// ---- analog_input/voltage/EL3164.TcPOU
(**
This function block abstracts the Beckhoff EtherCAT terminal EL3164 (0…10 V, 16 Bit)
*)
FUNCTION_BLOCK EL3164 IMPLEMENTS I_terminal_execution
VAR_INPUT
END_VAR
VAR_OUTPUT
	AI_Voltage_channel_1 		: I_AI_Voltage := _ar_channels[1];
	AI_Voltage_channel_2 		: I_AI_Voltage := _ar_channels[2];
	AI_Voltage_channel_3 		: I_AI_Voltage := _ar_channels[3];
	AI_Voltage_channel_4 		: I_AI_Voltage := _ar_channels[4];
	AI_percent_channe_1			: I_AI_percentage := _ar_channels[1];
	AI_percent_channe_2			: I_AI_percentage := _ar_channels[2];
	AI_percent_channe_3			: I_AI_percentage := _ar_channels[3];
	AI_percent_channe_4			: I_AI_percentage := _ar_channels[4];
END_VAR
VAR
// == IO Mapping ==============================================================
// The channel status Limits 1 and 2 have to be defined as BYTE since they are 
// of BIT2 in the terminal, but there is no such datatype in the PLC.

	WcState_WcState			AT%I*: BOOL;
	InfoData_State			AT%I*: UINT;
	InfoData_AdsAddr_netId  AT%I*: AMSNETID;
	InfoData_AdsAddr_port 	AT%I*: WORD;
	
	// Channel 1
	AI_Standard_Channel_1_Value        			AT%I*: INT;	
	AI_Standard_Channel_1_Status_Underrange   	AT%I*: BOOL;
	AI_Standard_Channel_1_Status_Overrange   	AT%I*: BOOL;
	AI_Standard_Channel_1_Status_Limit_1   		AT%I*: BYTE;
	AI_Standard_Channel_1_Status_Limit_2   		AT%I*: BYTE;
	AI_Standard_Channel_1_Status_Error   		AT%I*: BOOL;
	AI_Standard_Channel_1_Status_Sync_error   	AT%I*: BOOL;
	AI_Standard_Channel_1_Status_TxPDO_State   	AT%I*: BOOL;
	AI_Standard_Channel_1_Status_TxPDO_Toggle   AT%I*: BOOL;

	// Channel 2
	AI_Standard_Channel_2_Value        			AT%I*: INT;	
	AI_Standard_Channel_2_Status_Underrange   	AT%I*: BOOL;
	AI_Standard_Channel_2_Status_Overrange   	AT%I*: BOOL;
	AI_Standard_Channel_2_Status_Limit_1   		AT%I*: BYTE;
	AI_Standard_Channel_2_Status_Limit_2   		AT%I*: BYTE;
	AI_Standard_Channel_2_Status_Error   		AT%I*: BOOL;
	AI_Standard_Channel_2_Status_Sync_error   	AT%I*: BOOL;
	AI_Standard_Channel_2_Status_TxPDO_State   	AT%I*: BOOL;
	AI_Standard_Channel_2_Status_TxPDO_Toggle   AT%I*: BOOL;
	
	// Channel 3
	AI_Standard_Channel_3_Value        			AT%I*: INT;	
	AI_Standard_Channel_3_Status_Underrange   	AT%I*: BOOL;
	AI_Standard_Channel_3_Status_Overrange   	AT%I*: BOOL;
	AI_Standard_Channel_3_Status_Limit_1   		AT%I*: BYTE;
	AI_Standard_Channel_3_Status_Limit_2   		AT%I*: BYTE;
	AI_Standard_Channel_3_Status_Error   		AT%I*: BOOL;
	AI_Standard_Channel_3_Status_Sync_error   	AT%I*: BOOL;
	AI_Standard_Channel_3_Status_TxPDO_State   	AT%I*: BOOL;
	AI_Standard_Channel_3_Status_TxPDO_Toggle   AT%I*: BOOL;
	
	// Channel 4
	AI_Standard_Channel_4_Value        			AT%I*: INT;	
	AI_Standard_Channel_4_Status_Underrange   	AT%I*: BOOL;
	AI_Standard_Channel_4_Status_Overrange   	AT%I*: BOOL;
	AI_Standard_Channel_4_Status_Limit_1   		AT%I*: BYTE;  
	AI_Standard_Channel_4_Status_Limit_2   		AT%I*: BYTE;
	AI_Standard_Channel_4_Status_Error   		AT%I*: BOOL;
	AI_Standard_Channel_4_Status_Sync_error   	AT%I*: BOOL;
	AI_Standard_Channel_4_Status_TxPDO_State   	AT%I*: BOOL;
	AI_Standard_Channel_4_Status_TxPDO_Toggle   AT%I*: BOOL;
// ============================================================================

    _ar_channels : ARRAY[1..NUMBER_OF_CHANNELS] OF AI_Voltage_Channel[
		(adc_min:=ADC_MIN, adc_max:=ADC_MAX, physical_min:=PHYSICAL_MIN, physical_max:=PHYSICAL_MAX,channel_number:=1),
		(adc_min:=ADC_MIN, adc_max:=ADC_MAX, physical_min:=PHYSICAL_MIN, physical_max:=PHYSICAL_MAX,channel_number:=2),
		(adc_min:=ADC_MIN, adc_max:=ADC_MAX, physical_min:=PHYSICAL_MIN, physical_max:=PHYSICAL_MAX,channel_number:=3),
		(adc_min:=ADC_MIN, adc_max:=ADC_MAX, physical_min:=PHYSICAL_MIN, physical_max:=PHYSICAL_MAX,channel_number:=4)
    ];
    
	// ===============================================================================
	// CoE handling  
	// ==============
    _I_CoE_com_handler      : I_CoE_communication_handler;
    _CoE_prop_handler       : CoE_property_handler;
    // ====  CoE properties  ===========
	_p_DeviceName 			: CoE_property_string(Index:=16#1008 , SubIndex:=0, writable:=FALSE, propertyType:=0, pollingInterval:=T#5S);
	_p_DeviceType 			: CoE_property_udint(Index:=16#1000 , SubIndex:=0, writable:=FALSE, propertyType:=0, pollingInterval:=T#5S);
	_p_ProductCode 			: CoE_property_udint(Index:=16#1018 , SubIndex:=2, writable:=FALSE, propertyType:=0, pollingInterval:=T#5S);
	_p_Revision 			: CoE_property_udint(Index:=16#1018 , SubIndex:=3, writable:=FALSE, propertyType:=0, pollingInterval:=T#5S);
	_p_SerialNumber 		: CoE_property_udint(Index:=16#1018 , SubIndex:=4, writable:=FALSE, propertyType:=0, pollingInterval:=T#5S);
	_p_SoftwareVersion		: CoE_property_string(Index:=16#100A , SubIndex:=0, writable:=FALSE, propertyType:=0, pollingInterval:=T#5S);
	_p_VendorId 			: CoE_property_udint(Index:=16#1018 , SubIndex:=1, writable:=FALSE, propertyType:=0, pollingInterval:=T#5S);
	_p_HardwareVersion		: CoE_property_string(Index:=16#1009 , SubIndex:=0, writable:=FALSE, propertyType:=0, pollingInterval:=T#5S);
	// ==============
	_properties  : ARRAY[1..8]OF I_CoE_property:=[
		_p_DeviceName, _p_DeviceType, _p_ProductCode, _p_Revision, _p_SerialNumber, 
		_p_SoftwareVersion, _p_VendorId, _p_HardwareVersion
	];
	// ===============================================================================
    
    
	_I_InterfaceManager : I_InterfaceManager;
	_terminal_name      : STRING;
    errId               : HAL_ErrorEnum;
	_InitState          : INT;
    neg_wcState: f_trig;
    _j:INT;
	_terminal_id: UINT;

END_VAR
VAR CONSTANT
	ADC_MIN        	: INT:=0;
	ADC_MAX        	: INT:=32767;
	PHYSICAL_MIN 	: INT:=0;
	PHYSICAL_MAX 	: INT:=10;
	
    HARDWARE_REVSION : UINT:=19;
    NUMBER_OF_CHANNELS : INT:=4;
END_VAR


// Channel 1
_ar_channels[1].wcState							:= WcState_WcState;
_ar_channels[1].terminal_value                  := AI_Standard_Channel_1_Value;
_ar_channels[1].io_status_Underrange            := AI_Standard_Channel_1_Status_Underrange;
_ar_channels[1].io_status_Overrange             := AI_Standard_Channel_1_Status_Overrange;
_ar_channels[1].io_status_Limit_1_greater_value := AI_Standard_Channel_1_Status_Limit_1.0;
_ar_channels[1].io_status_Limit_1_smaller_value := AI_Standard_Channel_1_Status_Limit_1.1;
_ar_channels[1].io_status_Limit_2_greater_value := AI_Standard_Channel_1_Status_Limit_2.0;
_ar_channels[1].io_status_Limit_2_smaller_value := AI_Standard_Channel_1_Status_Limit_2.1;
_ar_channels[1].io_status_Error                 := AI_Standard_Channel_1_Status_Error;
_ar_channels[1].io_status_Sync_error            := AI_Standard_Channel_1_Status_Sync_error;
_ar_channels[1].io_status_TxPDO_State           := AI_Standard_Channel_1_Status_TxPDO_State;
_ar_channels[1].io_status_TxPDO_Toggle          := AI_Standard_Channel_1_Status_TxPDO_Toggle;

// Channel 2
_ar_channels[2].wcState                         := WcState_WcState;
_ar_channels[2].terminal_value                  := AI_Standard_Channel_2_Value;
_ar_channels[2].io_status_Underrange            := AI_Standard_Channel_2_Status_Underrange;
_ar_channels[2].io_status_Overrange             := AI_Standard_Channel_2_Status_Overrange;
_ar_channels[2].io_status_Limit_1_greater_value := AI_Standard_Channel_2_Status_Limit_1.0;
_ar_channels[2].io_status_Limit_1_smaller_value := AI_Standard_Channel_2_Status_Limit_1.1;
_ar_channels[2].io_status_Limit_2_greater_value := AI_Standard_Channel_2_Status_Limit_2.0;
_ar_channels[2].io_status_Limit_2_smaller_value := AI_Standard_Channel_2_Status_Limit_2.1;
_ar_channels[2].io_status_Error                 := AI_Standard_Channel_2_Status_Error;
_ar_channels[2].io_status_Sync_error            := AI_Standard_Channel_2_Status_Sync_error;
_ar_channels[2].io_status_TxPDO_State           := AI_Standard_Channel_2_Status_TxPDO_State;
_ar_channels[2].io_status_TxPDO_Toggle          := AI_Standard_Channel_2_Status_TxPDO_Toggle;

// Channel 3
_ar_channels[3].wcState                         := WcState_WcState;
_ar_channels[3].terminal_value                  := AI_Standard_Channel_3_Value;
_ar_channels[3].io_status_Underrange            := AI_Standard_Channel_3_Status_Underrange;
_ar_channels[3].io_status_Overrange             := AI_Standard_Channel_3_Status_Overrange;
_ar_channels[3].io_status_Limit_1_greater_value := AI_Standard_Channel_3_Status_Limit_1.0;
_ar_channels[3].io_status_Limit_1_smaller_value := AI_Standard_Channel_3_Status_Limit_1.1;
_ar_channels[3].io_status_Limit_2_greater_value := AI_Standard_Channel_3_Status_Limit_2.0;
_ar_channels[3].io_status_Limit_2_smaller_value := AI_Standard_Channel_3_Status_Limit_2.1;
_ar_channels[3].io_status_Error                 := AI_Standard_Channel_3_Status_Error;
_ar_channels[3].io_status_Sync_error            := AI_Standard_Channel_3_Status_Sync_error;
_ar_channels[3].io_status_TxPDO_State           := AI_Standard_Channel_3_Status_TxPDO_State;
_ar_channels[3].io_status_TxPDO_Toggle          := AI_Standard_Channel_3_Status_TxPDO_Toggle;

// Channel 4
_ar_channels[4].wcState                         := WcState_WcState;
_ar_channels[4].terminal_value                  := AI_Standard_Channel_4_Value;
_ar_channels[4].io_status_Underrange            := AI_Standard_Channel_4_Status_Underrange;
_ar_channels[4].io_status_Overrange             := AI_Standard_Channel_4_Status_Overrange;
_ar_channels[4].io_status_Limit_1_greater_value := AI_Standard_Channel_4_Status_Limit_1.0;
_ar_channels[4].io_status_Limit_1_smaller_value := AI_Standard_Channel_4_Status_Limit_1.1;
_ar_channels[4].io_status_Limit_2_greater_value := AI_Standard_Channel_4_Status_Limit_2.0;
_ar_channels[4].io_status_Limit_2_smaller_value := AI_Standard_Channel_4_Status_Limit_2.1;
_ar_channels[4].io_status_Error                 := AI_Standard_Channel_4_Status_Error;
_ar_channels[4].io_status_Sync_error            := AI_Standard_Channel_4_Status_Sync_error;
_ar_channels[4].io_status_TxPDO_State           := AI_Standard_Channel_4_Status_TxPDO_State;
_ar_channels[4].io_status_TxPDO_Toggle          := AI_Standard_Channel_4_Status_TxPDO_Toggle;


IF  _I_InterfaceManager <> 0 AND 
    _I_CoE_com_handler <> 0
THEN
    FOR _j:=1 TO NUMBER_OF_CHANNELS DO
        // should be possible to get rid of the address input 
        _ar_channels[_j](terminal_address:=InfoData_AdsAddr_port, CoE_communication_handler:=_I_CoE_com_handler);
    END_FOR
    
    _CoE_prop_handler(terminal_address:=InfoData_AdsAddr_port, CoE_communication_handler:=_I_CoE_com_handler, CoE_properties:=_properties);

    neg_wcState(CLK:=WcState_WcState);
    IF neg_wcState.Q THEN
        ;
    END_IF
END_IF

METHOD FB_init : BOOL
VAR_INPUT
	bInitRetains : BOOL; // if TRUE, the retain variables are initialized (warm start / cold start)
	bInCopyCode : BOOL;  // if TRUE, the instance afterwards gets moved into the copy code (online change)
	CoE_communication_handler   : I_CoE_communication_handler;
	InterfaceManager            : I_InterfaceManager;
	name                        : STRING;
END_VAR

_I_CoE_com_handler := CoE_communication_handler;

FOR _j:=1 TO NUMBER_OF_CHANNELS DO
    _ar_channels[_j].CoE_communication_handler := CoE_communication_handler;
END_FOR

_terminal_name := name;
_I_InterfaceManager := InterfaceManager;

// register  terminal and all channel interfaces
IF InterfaceManager <> 0 THEN
    _I_InterfaceManager.register_terminal(terminal_name:=_terminal_name , errId=>errId , terminalId=>_terminal_id);
    
    FOR _j:=1 TO NUMBER_OF_CHANNELS DO
        _ar_channels[_j].register_channel(terminalId:=_terminal_id , I_interface_manager:=_I_InterfaceManager , errId=>errId );
        IF errId <> HAL_ErrorEnum.no_error THEN
            ;  // ToDo: add logging or Error handling 
        END_IF 
    END_FOR
END_IF
END_METHOD

METHOD run : BOOL
THIS^();
END_METHOD

END_FUNCTION_BLOCK

// ---- analog_input/_internal/AI_Voltage_Channel.TcPOU
FUNCTION_BLOCK AI_Voltage_Channel IMPLEMENTS I_AI_Voltage, I_AI_percentage
VAR_INPUT
	terminal_address		    : WORD;
	CoE_communication_handler	: I_CoE_communication_handler;
END_VAR
VAR_OUTPUT
END_VAR
VAR
	_adc_min        : INT;
    _adc_max        : INT;
	_physical_min 	: INT;
	_physical_max 	: INT;
	_channel_number : UsINT;
	_rValue			: REAL;
	_wcState		: BOOL;
	
	// ===============================================================================
	// CoE handling  
    // ==============
    _CoE_prop_handler      : CoE_property_handler;
    _CoE_channel_offset     : INT;
    index_1 				: WORD:= 16#8000 + INT_TO_WORD(_CoE_channel_offset);	
    // ====  CoE properties  ===========
	_p_Enable_user_scale    		: CoE_property_bool(Index:=index_1 , SubIndex:=1, writable:=TRUE, propertyType:=0, pollingInterval:=T#5S);
	_p_Presentation 				: CoE_property_usint(Index:=index_1 , SubIndex:=2, writable:=TRUE, propertyType:=0, pollingInterval:=T#5S);			// DT0800EN03
	_p_Watchdog 					: CoE_property_usint(Index:=index_1 , SubIndex:=5, writable:=TRUE, propertyType:=0, pollingInterval:=T#5S);			// DT0801EN02
	_p_Enable_user_calibration  	: CoE_property_bool(Index:=index_1 , SubIndex:=7, writable:=TRUE, propertyType:=0, pollingInterval:=T#5S);
	_p_Enable_vendor_calibration    : CoE_property_bool(Index:=index_1 , SubIndex:=8, writable:=TRUE, propertyType:=0, pollingInterval:=T#5S);
	_p_Offset   					: CoE_property_int(Index:=index_1 , SubIndex:=17, writable:=TRUE, propertyType:=0, pollingInterval:=T#5S);
	_p_Gain 						: CoE_property_dint(Index:=index_1 , SubIndex:=18, writable:=TRUE, propertyType:=0, pollingInterval:=T#5S);
	_p_Default_output   			: CoE_property_int(Index:=index_1 , SubIndex:=19, writable:=TRUE, propertyType:=0, pollingInterval:=T#5S);
	_p_Default_output_ramp  		: CoE_property_uint(Index:=index_1 , SubIndex:=20, writable:=TRUE, propertyType:=0, pollingInterval:=T#5S);
	_p_User_calibration_offset  	: CoE_property_int(Index:=index_1 , SubIndex:=21, writable:=TRUE, propertyType:=0, pollingInterval:=T#5S);
	_p_User_calibration_gain    	: CoE_property_uint(Index:=index_1 , SubIndex:=22, writable:=TRUE, propertyType:=0, pollingInterval:=T#5S);
	// ==============
	_properties  : ARRAY[1..11]OF I_CoE_property:=[
		_p_Enable_user_scale, _p_Presentation, _p_Watchdog, _p_Enable_user_calibration, _p_Enable_vendor_calibration, _p_Offset,
		_p_Gain, _p_Default_output, _p_Default_output_ramp, _p_User_calibration_offset, _p_User_calibration_gain];
	// ===============================================================================


	//  ====  I_AI_percentage  ====
	_max_value 	: REAL:=10.0;
	_min_value 	: REAL:=0.0;
	_value: REAL;
	
	_errId: HAL_ErrorEnum;
	neg_wcState: f_trig;
END_VAR

// CoE Property handling 
_CoE_prop_handler(terminal_address:=terminal_address, CoE_communication_handler:=CoE_communication_handler, CoE_properties:=_properties);

neg_wcState(CLK:=_wcState);
IF neg_wcState.Q THEN
    ;
END_IF

PROPERTY errId : HAL_ErrorEnum
GET
errId := _errId;
END_GET
END_PROPERTY

METHOD FB_init : BOOL
VAR_INPUT
	bInitRetains 	: BOOL; // if TRUE, the retain variables are initialized (warm start / cold start)
	bInCopyCode 	: BOOL;  // if TRUE, the instance afterwards gets moved into the copy code (online change)
    adc_min         : INT;
    adc_max         : INT;
	physical_min 	: INT;
	physical_max 	: INT;
	channel_number  : UsINT;
END_VAR

VAR
	i: UINT;
END_VAR

_adc_min        := adc_min;
_adc_max        := adc_max;
_physical_min 	:= physical_min;
_physical_max 	:= physical_max;
_channel_number :=channel_number;

CASE channel_number OF
	1:
		_CoE_channel_offset:=16#0;
	2:
		_CoE_channel_offset:=16#10;
	3:
		_CoE_channel_offset:=16#20;
	4:
		_CoE_channel_offset:=16#30;
END_CASE
END_METHOD

METHOD get_Default_output : BOOL
VAR_OUTPUT
	value	: INT;
END_VAR
get_Default_output:=_p_Default_output.get_value(value=>value, errId => );
END_METHOD

METHOD get_Default_output_ramp : BOOL
VAR_OUTPUT
	value	: UINT;
END_VAR
get_Default_output_ramp:=_p_Default_output_ramp.get_value(value=>value, errId => );
END_METHOD

METHOD get_Enable_user_calibration : BOOL
VAR_OUTPUT
	value	: BOOL;
END_VAR
get_Enable_user_calibration:=_p_Enable_user_calibration.get_value(value=>value, errId => );
END_METHOD

METHOD get_Enable_user_scale : BOOL
VAR_OUTPUT
	value	: BOOL;
END_VAR
get_Enable_user_scale:=_p_Enable_user_scale.get_value(value=>value, errId => );
END_METHOD

METHOD get_Enable_vendor_calibration : BOOL
VAR_OUTPUT
	value	: BOOL;
END_VAR
get_Enable_vendor_calibration:=_p_Enable_vendor_calibration.get_value(value=>value, errId => );
END_METHOD

METHOD get_Gain : BOOL
VAR_OUTPUT
	value	: DINT;
END_VAR
get_Gain:=_p_Gain.get_value(value=>value, errId => );
END_METHOD

METHOD get_Offset : BOOL
VAR_OUTPUT
	value	: INT;
END_VAR
get_Offset:=_p_Offset.get_value(value=>value, errId => );
END_METHOD

METHOD get_Presentation : BOOL
VAR_OUTPUT
	value	: ENU_DT0801EN03;
END_VAR

VAR
	tmp: USINT;
END_VAR
get_Presentation:=_p_Presentation.get_value(value=>tmp, errId => );
value:=USINT_TO_INT(tmp);
END_METHOD

METHOD get_User_calibration_gain : BOOL
VAR_OUTPUT
	value	: UINT;
END_VAR
get_User_calibration_gain:=_p_User_calibration_gain.get_value(value=>value, errId => );
END_METHOD

METHOD get_User_calibration_offset : BOOL
VAR_OUTPUT
	value	: INT;
END_VAR
get_User_calibration_offset:=_p_User_calibration_offset.get_value(value=>value, errId => );
END_METHOD

METHOD get_Watchdog : BOOL
VAR_OUTPUT
	value	: ENU_DT0800EN02;
END_VAR

VAR
	tmp: USINT;
END_VAR
get_Watchdog:=_p_Watchdog.get_value(value=>tmp, errId => );
value := USINT_TO_INT(tmp);
END_METHOD

PROPERTY io_status_Error : bool
GET
END_GET
SET
END_SET
END_PROPERTY

PROPERTY io_status_Limit_1_greater_value : bool
GET
END_GET
SET
END_SET
END_PROPERTY

PROPERTY io_status_Limit_1_smaller_value : bool
GET
END_GET
SET
END_SET
END_PROPERTY

PROPERTY io_status_Limit_2_greater_value : bool
GET
END_GET
SET
END_SET
END_PROPERTY

PROPERTY io_status_Limit_2_smaller_value : bool
GET
END_GET
SET
END_SET
END_PROPERTY

PROPERTY io_status_Overrange : bool
GET
END_GET
SET
END_SET
END_PROPERTY

PROPERTY io_status_Sync_error : bool
GET
END_GET
SET
END_SET
END_PROPERTY

PROPERTY io_status_TxPDO_State : bool
GET
END_GET
SET
END_SET
END_PROPERTY

PROPERTY io_status_TxPDO_Toggle : bool
GET
END_GET
SET
END_SET
END_PROPERTY

PROPERTY io_status_Underrange : bool
GET
END_GET
SET
END_SET
END_PROPERTY

PROPERTY max_value : REAL
GET
max_value := _max_value;
END_GET
SET
IF max_value <= 0 THEN
	_max_value := 0.0001;
ELSE
	_max_value := max_value;
END_IF
END_SET
END_PROPERTY

PROPERTY min_value : REAL
GET
min_value := _min_value;
END_GET
SET
_min_value := min_value;
END_SET
END_PROPERTY

METHOD register_channel : BOOL
VAR_INPUT
    terminalId : UINT;
    I_interface_manager : I_interfaceManager;
END_VAR
VAR_OUTPUT
	errId		: HAL_ErrorEnum;
END_VAR
THIS^.register_I_AI_percentage(terminalId:=terminalId , I_interface_manager:=I_interface_manager , errId=>errId );
IF errId = HAL_ErrorEnum.no_error THEN
	THIS^.register_I_AI_Voltage(terminalId:=terminalId , I_interface_manager:=I_interface_manager , errId=>errId );
END_IF
END_METHOD

METHOD register_I_AI_percentage : BOOL
VAR_INPUT
    terminalId : UINT;
    I_interface_manager : I_interfaceManager;
END_VAR
VAR_OUTPUT
	errId		: HAL_ErrorEnum;
END_VAR
register_I_AI_percentage:= I_interface_manager.register_I_AI_Percentage(THIS^, terminalId, channel_number := THIS^._channel_number, errId=>errId);
END_METHOD

METHOD register_I_AI_Voltage : BOOL
VAR_INPUT
    terminalId : UINT;
    I_interface_manager : I_interfaceManager;
END_VAR
VAR_OUTPUT
	errId		: HAL_ErrorEnum;
END_VAR
register_I_AI_Voltage:= I_interface_manager.register_I_AI_Voltage(THIS^, terminalId, channel_number := THIS^._channel_number, errId=>errId);
END_METHOD

PROPERTY rValue : REAL
GET
rValue:=_rValue;
END_GET
SET
IF rValue < DINT_TO_REAL(_physical_min) THEN
	_errId := 6;
ELSIF rValue > DINT_TO_REAL(_physical_max) THEN
	_errId := 7;
ELSE
	_rValue := rValue;
END_IF
END_SET
END_PROPERTY

METHOD set_Default_output : BOOL
VAR_INPUT
	value	: INT;
END_VAR
set_Default_output:=_p_Default_output.set_value(value:=value);
END_METHOD

METHOD set_Default_output_ramp : BOOL
VAR_INPUT
	value	: UINT;
END_VAR
set_Default_output_ramp:=_p_Default_output_ramp.set_value(value:=value);
END_METHOD

METHOD set_Enable_user_calibration : BOOL
VAR_INPUT
	value	: BOOL;
END_VAR
set_Enable_user_calibration:=_p_Enable_user_calibration.set_value(value:=value);
END_METHOD

METHOD set_Enable_user_scale : BOOL
VAR_INPUT
	value	: BOOL;
END_VAR
set_Enable_user_scale:=_p_Enable_user_scale.set_value(value:=value);
END_METHOD

METHOD set_Enable_vendor_calibration : BOOL
VAR_INPUT
	value	: BOOL;
END_VAR
set_Enable_vendor_calibration:=_p_Enable_vendor_calibration.set_value(value:=value);
END_METHOD

METHOD set_Gain : BOOL
VAR_INPUT
	value	: DINT;
END_VAR
set_Gain:=_p_Gain.set_value(value:=value);
END_METHOD

METHOD set_Offset : BOOL
VAR_INPUT
	value	: INT;
END_VAR
set_Offset:=_p_Offset.set_value(value:=value);
END_METHOD

METHOD set_Presentation : BOOL
VAR_INPUT
	value	: ENU_DT0801EN03;
END_VAR
set_Presentation:=_p_Presentation.set_value(value:=INT_TO_USINT(value));
END_METHOD

METHOD set_User_calibration_gain : BOOL
VAR_INPUT
	value	: UINT;
END_VAR
set_User_calibration_gain:=_p_User_calibration_gain.set_value(value:=value);
END_METHOD

METHOD set_User_calibration_offset : BOOL
VAR_INPUT
	value	: INT;
END_VAR
set_User_calibration_offset:=_p_User_calibration_offset.set_value(value:=value);
END_METHOD

METHOD set_Watchdog : BOOL
VAR_INPUT
	value	: ENU_DT0800EN02;
END_VAR
set_Watchdog:=_p_Watchdog.set_value(value:=int_TO_USINT(value));
END_METHOD

PROPERTY terminal_value : int
SET
linear_adc_to_phy(
	physical_min	:= _physical_min, 
	physical_max	:= _physical_max, 
	adc_min			:= _adc_min, 
	adc_max			:= _adc_max, 
	adc_value		:= terminal_value, 
	physical_value	=> _rValue, 
	errId			=> _errId
);

linear_adc_to_phy(
	physical_min	:= 0, 
	physical_max	:= 100, 
	adc_min			:= REAL_TO_DINT(_min_value), 
	adc_max			:= REAL_TO_DINT(_max_value), 
	adc_value		:= REAL_TO_DINT(_rValue), 
	physical_value	=> _value, 
	errId			=> _errId
);
END_SET
END_PROPERTY

PROPERTY value : REAL
GET
value := _value;
END_GET
END_PROPERTY

PROPERTY wcState : bool
GET
wcState:=_wcState;
END_GET
SET
_wcState:=wcState;
END_SET
END_PROPERTY

END_FUNCTION_BLOCK

// ---- analog_input/temperature/EL3202_0010.TcPOU
FUNCTION_BLOCK EL3202_0010 IMPLEMENTS I_terminal_execution
VAR_INPUT
END_VAR
VAR_OUTPUT
    AI_Temperature_channel_1 	: I_AI_Temperature := _ar_channels[1];
	AI_Temperature_channel_2 	: I_AI_Temperature := _ar_channels[2];
	AI_percent_channe_1			: I_AI_percentage := _ar_channels[1];
	AI_percent_channe_2			: I_AI_percentage := _ar_channels[2];
END_VAR
VAR
// == IO Mapping ==============================================================
	WcState_WcState			AT%I*: BOOL;
	InfoData_State			AT%I*: UINT;
	InfoData_AdsAddr_netId  AT%I*: AMSNETID;
	InfoData_AdsAddr_port 	AT%I*: WORD;
	
	// Channel 1
	RTD_Inputs_Channel_1_Value        			AT%I*: INT;	
	RTD_Inputs_Channel_1_Status_Underrange   	AT%I*: BOOL;
	RTD_Inputs_Channel_1_Status_Overrange   	AT%I*: BOOL;
	RTD_Inputs_Channel_1_Status_Limit_1   		AT%I*: BYTE;
	RTD_Inputs_Channel_1_Status_Limit_2   		AT%I*: BYTE;
	RTD_Inputs_Channel_1_Status_Error   		AT%I*: BOOL;
	RTD_Inputs_Channel_1_Status_TxPDO_State   	AT%I*: BOOL;
	RTD_Inputs_Channel_1_Status_TxPDO_Toggle   	AT%I*: BOOL;
	
	// Channel 2
	RTD_Inputs_Channel_2_Value        			AT%I*: INT;	
	RTD_Inputs_Channel_2_Status_Underrange   	AT%I*: BOOL;
	RTD_Inputs_Channel_2_Status_Overrange   	AT%I*: BOOL;
	RTD_Inputs_Channel_2_Status_Limit_1   		AT%I*: BYTE;
	RTD_Inputs_Channel_2_Status_Limit_2   		AT%I*: BYTE;
	RTD_Inputs_Channel_2_Status_Error   		AT%I*: BOOL;
	RTD_Inputs_Channel_2_Status_TxPDO_State   	AT%I*: BOOL;
	RTD_Inputs_Channel_2_Status_TxPDO_Toggle   	AT%I*: BOOL;
// ============================================================================

    _ar_channels : ARRAY[1..NUMBER_OF_CHANNELS] OF AI_Temperature_Channel[
		(adc_min:=ADC_MIN, adc_max:=ADC_MAX, physical_min:=PHYSICAL_MIN, physical_max:=PHYSICAL_MAX,channel_number:=1),
		(adc_min:=ADC_MIN, adc_max:=ADC_MAX, physical_min:=PHYSICAL_MIN, physical_max:=PHYSICAL_MAX,channel_number:=2)
    ];
    
	// ===============================================================================
	// CoE handling  
	// ==============
    _I_CoE_com_handler      : I_CoE_communication_handler;
    _CoE_prop_handler       : CoE_property_handler;
    // ====  CoE properties  ===========
	_p_DeviceName 			: CoE_property_string(Index:=16#1008 , SubIndex:=0, writable:=FALSE, propertyType:=0, pollingInterval:=T#5S);
	_p_DeviceType 			: CoE_property_udint(Index:=16#1000 , SubIndex:=0, writable:=FALSE, propertyType:=0, pollingInterval:=T#5S);
	_p_ProductCode 			: CoE_property_udint(Index:=16#1018 , SubIndex:=2, writable:=FALSE, propertyType:=0, pollingInterval:=T#5S);
	_p_Revision 			: CoE_property_udint(Index:=16#1018 , SubIndex:=3, writable:=FALSE, propertyType:=0, pollingInterval:=T#5S);
	_p_SerialNumber 		: CoE_property_udint(Index:=16#1018 , SubIndex:=4, writable:=FALSE, propertyType:=0, pollingInterval:=T#5S);
	_p_SoftwareVersion		: CoE_property_string(Index:=16#100A , SubIndex:=0, writable:=FALSE, propertyType:=0, pollingInterval:=T#5S);
	_p_VendorId 			: CoE_property_udint(Index:=16#1018 , SubIndex:=1, writable:=FALSE, propertyType:=0, pollingInterval:=T#5S);
	_p_HardwareVersion		: CoE_property_string(Index:=16#1009 , SubIndex:=0, writable:=FALSE, propertyType:=0, pollingInterval:=T#5S);
	// ==============
	_properties  : ARRAY[1..8]OF I_CoE_property:=[
		_p_DeviceName, _p_DeviceType, _p_ProductCode, _p_Revision, _p_SerialNumber, 
		_p_SoftwareVersion, _p_VendorId, _p_HardwareVersion
	];
	// ===============================================================================
    
	_I_InterfaceManager : I_InterfaceManager;
	_terminal_name      : STRING;
    _terminal_id        : UINT;
    errId               : HAL_ErrorEnum;
	_InitState          : INT;
    neg_wcState : f_trig;
	_j      : USINT;
END_VAR
VAR CONSTANT
	ADC_MIN        	: INT:=0;
	ADC_MAX        	: INT:=32767;
	PHYSICAL_MIN 	: INT:=0;
	PHYSICAL_MAX 	: INT:=10;
	
    HARDWARE_REVSION : UINT:=19;
    NUMBER_OF_CHANNELS : USINT:=2;
END_VAR


// Channel 1
_ar_channels[1].wcState							:= WcState_WcState;
_ar_channels[1].terminal_value 					:= RTD_Inputs_Channel_1_Value;
_ar_channels[1].io_status_Underrange 			:= RTD_Inputs_Channel_1_Status_Underrange;
_ar_channels[1].io_status_Overrange 			:= RTD_Inputs_Channel_1_Status_Overrange;
_ar_channels[1].io_status_Limit_1_greater_value := RTD_Inputs_Channel_1_Status_Limit_1.0;
_ar_channels[1].io_status_Limit_1_smaller_value	:= RTD_Inputs_Channel_1_Status_Limit_1.1;
_ar_channels[1].io_status_Limit_2_greater_value := RTD_Inputs_Channel_1_Status_Limit_2.0;
_ar_channels[1].io_status_Limit_2_smaller_value	:= RTD_Inputs_Channel_1_Status_Limit_2.1;
_ar_channels[1].io_status_Error 				:= RTD_Inputs_Channel_1_Status_Error;
_ar_channels[1].io_status_TxPDO_State 			:= RTD_Inputs_Channel_1_Status_TxPDO_State;
_ar_channels[1].io_status_TxPDO_Toggle 			:= RTD_Inputs_Channel_1_Status_TxPDO_Toggle;

// Channel 2
_ar_channels[2].wcState							:= WcState_WcState;
_ar_channels[2].terminal_value 					:= RTD_Inputs_Channel_2_Value;
_ar_channels[2].io_status_Underrange 			:= RTD_Inputs_Channel_2_Status_Underrange;
_ar_channels[2].io_status_Overrange 			:= RTD_Inputs_Channel_2_Status_Overrange;
_ar_channels[2].io_status_Limit_1_greater_value := RTD_Inputs_Channel_2_Status_Limit_1.0;
_ar_channels[2].io_status_Limit_1_smaller_value	:= RTD_Inputs_Channel_2_Status_Limit_1.1;
_ar_channels[2].io_status_Limit_2_greater_value := RTD_Inputs_Channel_2_Status_Limit_2.0;
_ar_channels[2].io_status_Limit_2_smaller_value	:= RTD_Inputs_Channel_2_Status_Limit_2.1;
_ar_channels[2].io_status_Error 				:= RTD_Inputs_Channel_2_Status_Error;
_ar_channels[2].io_status_TxPDO_State 			:= RTD_Inputs_Channel_2_Status_TxPDO_State;
_ar_channels[2].io_status_TxPDO_Toggle 			:= RTD_Inputs_Channel_2_Status_TxPDO_Toggle;


IF  _I_InterfaceManager <> 0 AND 
    _I_CoE_com_handler <> 0
THEN
    FOR _j:=1 TO NUMBER_OF_CHANNELS DO
        // should be possible to get rid of the address input 
        _ar_channels[_j](terminal_address:=InfoData_AdsAddr_port, CoE_communication_handler:=_I_CoE_com_handler);
    END_FOR
    
    _CoE_prop_handler(terminal_address:=InfoData_AdsAddr_port, CoE_communication_handler:=_I_CoE_com_handler, CoE_properties:=_properties);

    neg_wcState(CLK:=WcState_WcState);
    IF neg_wcState.Q THEN
        ;
    END_IF
END_IF

METHOD FB_init : BOOL
VAR_INPUT
	bInitRetains : BOOL; // if TRUE, the retain variables are initialized (warm start / cold start)
	bInCopyCode : BOOL;  // if TRUE, the instance afterwards gets moved into the copy code (online change)
	CoE_communication_handler   : I_CoE_communication_handler;
    InterfaceManager            : I_InterfaceManager;
	name                        : STRING;
END_VAR

_I_CoE_com_handler := CoE_communication_handler;

FOR _j:=1 TO NUMBER_OF_CHANNELS DO
    _ar_channels[_j].CoE_communication_handler := CoE_communication_handler;
END_FOR

_terminal_name := name;
_I_InterfaceManager := InterfaceManager;

// register  terminal and all channel interfaces
IF InterfaceManager <> 0 THEN
    _I_InterfaceManager.register_terminal(terminal_name:=_terminal_name , errId=>errId , terminalId=>_terminal_id);
    
    FOR _j:=1 TO NUMBER_OF_CHANNELS DO
        _ar_channels[_j].register_channel(terminalId:=_terminal_id , I_interface_manager:=_I_InterfaceManager , errId=>errId );
        IF errId <> HAL_ErrorEnum.no_error THEN
            ;  // ToDo: add logging or Error handling 
        END_IF 
    END_FOR
END_IF
END_METHOD

METHOD run : BOOL
THIS^();
END_METHOD

END_FUNCTION_BLOCK

// ---- analog_input/_internal/AI_Temperature_Channel.TcPOU
FUNCTION_BLOCK AI_Temperature_Channel IMPLEMENTS I_terminal_channel, I_AI_Temperature, I_AI_percentage
VAR_INPUT
	terminal_address		: WORD;
	CoE_communication_handler	: I_CoE_communication_handler;
END_VAR
VAR_OUTPUT
END_VAR
VAR
	_adc_min        : INT;
    _adc_max        : INT;
	_physical_min 	: INT;
	_physical_max 	: INT;
	_channel_number : USINT;
	_rValue			: REAL;
	_wcState		: BOOL;
	
	// ===============================================================================
	// CoE handling  
    // ==============
    _CoE_prop_handler      : CoE_property_handler;
    _CoE_channel_offset     : INT;
    index_1 				: WORD:= 16#8000 + INT_TO_WORD(_CoE_channel_offset);	
    // ====  CoE properties  ===========
	_p_Enable_user_scale    		: CoE_property_bool(Index:=index_1 , SubIndex:=1, writable:=TRUE, propertyType:=0, pollingInterval:=T#5S);
	_p_Presentation 				: CoE_property_usint(Index:=index_1 , SubIndex:=2, writable:=TRUE, propertyType:=0, pollingInterval:=T#5S);			// DT0800EN03
	_p_Watchdog 					: CoE_property_usint(Index:=index_1 , SubIndex:=5, writable:=TRUE, propertyType:=0, pollingInterval:=T#5S);			// DT0801EN02
	_p_Enable_user_calibration  	: CoE_property_bool(Index:=index_1 , SubIndex:=7, writable:=TRUE, propertyType:=0, pollingInterval:=T#5S);
	_p_Enable_vendor_calibration    : CoE_property_bool(Index:=index_1 , SubIndex:=8, writable:=TRUE, propertyType:=0, pollingInterval:=T#5S);
	_p_Offset   					: CoE_property_int(Index:=index_1 , SubIndex:=17, writable:=TRUE, propertyType:=0, pollingInterval:=T#5S);
	_p_Gain 						: CoE_property_dint(Index:=index_1 , SubIndex:=18, writable:=TRUE, propertyType:=0, pollingInterval:=T#5S);
	_p_Default_output   			: CoE_property_int(Index:=index_1 , SubIndex:=19, writable:=TRUE, propertyType:=0, pollingInterval:=T#5S);
	_p_Default_output_ramp  		: CoE_property_uint(Index:=index_1 , SubIndex:=20, writable:=TRUE, propertyType:=0, pollingInterval:=T#5S);
	_p_User_calibration_offset  	: CoE_property_int(Index:=index_1 , SubIndex:=21, writable:=TRUE, propertyType:=0, pollingInterval:=T#5S);
	_p_User_calibration_gain    	: CoE_property_uint(Index:=index_1 , SubIndex:=22, writable:=TRUE, propertyType:=0, pollingInterval:=T#5S);
	// ==============
	_properties  : ARRAY[1..11]OF I_CoE_property:=[
		_p_Enable_user_scale, _p_Presentation, _p_Watchdog, _p_Enable_user_calibration, _p_Enable_vendor_calibration, _p_Offset,
		_p_Gain, _p_Default_output, _p_Default_output_ramp, _p_User_calibration_offset, _p_User_calibration_gain];
	// ===============================================================================
    
	
	//  ====  I_AI_percentage  ====
	_max_value 	: REAL:=10.0;
	_min_value 	: REAL:=0.0;
	_value: REAL;
	
	_errId: HAL_ErrorEnum;
    neg_wcState: f_trig;
END_VAR

// CoE Property handling 
_CoE_prop_handler(terminal_address:=terminal_address, CoE_communication_handler:=CoE_communication_handler, CoE_properties:=_properties);

neg_wcState(CLK:=_wcState);
IF neg_wcState.Q THEN
    ;
END_IF

PROPERTY errId : HAL_ErrorEnum
GET
errId := _errId;
END_GET
END_PROPERTY

METHOD FB_init : BOOL
VAR_INPUT
	bInitRetains 	: BOOL; // if TRUE, the retain variables are initialized (warm start / cold start)
	bInCopyCode 	: BOOL;  // if TRUE, the instance afterwards gets moved into the copy code (online change)
    adc_min         : INT;
    adc_max         : INT;
	physical_min 	: INT;
	physical_max 	: INT;
	channel_number  : USINT;
END_VAR

VAR
	i: UINT;
END_VAR

_adc_min        := adc_min;
_adc_max        := adc_max;
_physical_min 	:= physical_min;
_physical_max 	:= physical_max;
_channel_number :=channel_number;

CASE channel_number OF
	1:
		_CoE_channel_offset:=16#0;
	2:
		_CoE_channel_offset:=16#10;
	3:
		_CoE_channel_offset:=16#20;
	4:
		_CoE_channel_offset:=16#30;
END_CASE
END_METHOD

METHOD get_Default_output : BOOL
VAR_OUTPUT
	value	: INT;
END_VAR
get_Default_output:=_p_Default_output.get_value(value=>value, errId => );
END_METHOD

METHOD get_Default_output_ramp : BOOL
VAR_OUTPUT
	value	: UINT;
END_VAR
get_Default_output_ramp:=_p_Default_output_ramp.get_value(value=>value, errId => );
END_METHOD

METHOD get_Enable_user_calibration : BOOL
VAR_OUTPUT
	value	: BOOL;
END_VAR
get_Enable_user_calibration:=_p_Enable_user_calibration.get_value(value=>value, errId => );
END_METHOD

METHOD get_Enable_user_scale : BOOL
VAR_OUTPUT
	value	: BOOL;
END_VAR
get_Enable_user_scale:=_p_Enable_user_scale.get_value(value=>value, errId => );
END_METHOD

METHOD get_Enable_vendor_calibration : BOOL
VAR_OUTPUT
	value	: BOOL;
END_VAR
get_Enable_vendor_calibration:=_p_Enable_vendor_calibration.get_value(value=>value, errId => );
END_METHOD

METHOD get_Gain : BOOL
VAR_OUTPUT
	value	: DINT;
END_VAR
get_Gain:=_p_Gain.get_value(value=>value, errId => );
END_METHOD

METHOD get_Offset : BOOL
VAR_OUTPUT
	value	: INT;
END_VAR
get_Offset:=_p_Offset.get_value(value=>value, errId => );
END_METHOD

METHOD get_Presentation : BOOL
VAR_OUTPUT
	value	: ENU_DT0801EN03;
END_VAR

VAR
	tmp: USINT;
END_VAR
get_Presentation:=_p_Presentation.get_value(value=>tmp, errId => );
value:=USINT_TO_INT(tmp);
END_METHOD

METHOD get_User_calibration_gain : BOOL
VAR_OUTPUT
	value	: UINT;
END_VAR
get_User_calibration_gain:=_p_User_calibration_gain.get_value(value=>value, errId => );
END_METHOD

METHOD get_User_calibration_offset : BOOL
VAR_OUTPUT
	value	: INT;
END_VAR
get_User_calibration_offset:=_p_User_calibration_offset.get_value(value=>value, errId => );
END_METHOD

METHOD get_Watchdog : BOOL
VAR_OUTPUT
	value	: ENU_DT0800EN02;
END_VAR

VAR
	tmp: USINT;
END_VAR
get_Watchdog:=_p_Watchdog.get_value(value=>tmp, errId => );
value := USINT_TO_INT(tmp);
END_METHOD

PROPERTY io_status_Error : bool
GET
END_GET
SET
END_SET
END_PROPERTY

PROPERTY io_status_Limit_1_greater_value : bool
GET
END_GET
SET
END_SET
END_PROPERTY

PROPERTY io_status_Limit_1_smaller_value : bool
GET
END_GET
SET
END_SET
END_PROPERTY

PROPERTY io_status_Limit_2_greater_value : bool
GET
END_GET
SET
END_SET
END_PROPERTY

PROPERTY io_status_Limit_2_smaller_value : bool
GET
END_GET
SET
END_SET
END_PROPERTY

PROPERTY io_status_Overrange : bool
GET
END_GET
SET
END_SET
END_PROPERTY

PROPERTY io_status_Sync_error : bool
GET
END_GET
SET
END_SET
END_PROPERTY

PROPERTY io_status_TxPDO_State : bool
GET
END_GET
SET
END_SET
END_PROPERTY

PROPERTY io_status_TxPDO_Toggle : bool
GET
END_GET
SET
END_SET
END_PROPERTY

PROPERTY io_status_Underrange : bool
GET
END_GET
SET
END_SET
END_PROPERTY

PROPERTY max_value : REAL
GET
max_value := _max_value;
END_GET
SET
IF max_value <= 0 THEN
	_max_value := 0.0001;
ELSE
	_max_value := max_value;
END_IF
END_SET
END_PROPERTY

PROPERTY min_value : REAL
GET
min_value := _min_value;
END_GET
SET
_min_value := min_value;
END_SET
END_PROPERTY

METHOD register_channel : BOOL
VAR_INPUT
    terminalId : UINT;
    I_interface_manager : I_interfaceManager;
END_VAR
VAR_OUTPUT
	errId		: HAL_ErrorEnum;
END_VAR
THIS^.register_I_AI_percentage(terminalId:=terminalId , I_interface_manager:=I_interface_manager , errId=>errId );
IF errId = HAL_ErrorEnum.no_error THEN
	THIS^.register_I_AI_Temperature(terminalId:=terminalId , I_interface_manager:=I_interface_manager , errId=>errId );
END_IF
END_METHOD

METHOD register_I_AI_percentage : BOOL
VAR_INPUT
    terminalId : UINT;
    I_interface_manager : I_interfaceManager;
END_VAR
VAR_OUTPUT
	errId		: HAL_ErrorEnum;
END_VAR
register_I_AI_percentage:= I_interface_manager.register_I_AI_Percentage(THIS^, terminalId, channel_number := THIS^._channel_number, errId=>errId);
END_METHOD

METHOD register_I_AI_Temperature : BOOL
VAR_INPUT
    terminalId : UINT;
    I_interface_manager : I_interfaceManager;
END_VAR
VAR_OUTPUT
	errId		: HAL_ErrorEnum;
END_VAR
register_I_AI_Temperature:= I_interface_manager.register_I_AI_Temperature(THIS^, terminalId, channel_number := THIS^._channel_number, errId=>errId);
END_METHOD

PROPERTY rValue : REAL
GET
rValue:=_rValue;
END_GET
SET
IF rValue < DINT_TO_REAL(_physical_min) THEN
	_errId := 6;
ELSIF rValue > DINT_TO_REAL(_physical_max) THEN
	_errId := 7;
ELSE
	_rValue := rValue;
END_IF
END_SET
END_PROPERTY

METHOD set_Default_output : BOOL
VAR_INPUT
	value	: INT;
END_VAR
set_Default_output:=_p_Default_output.set_value(value:=value);
END_METHOD

METHOD set_Default_output_ramp : BOOL
VAR_INPUT
	value	: UINT;
END_VAR
set_Default_output_ramp:=_p_Default_output_ramp.set_value(value:=value);
END_METHOD

METHOD set_Enable_user_calibration : BOOL
VAR_INPUT
	value	: BOOL;
END_VAR
set_Enable_user_calibration:=_p_Enable_user_calibration.set_value(value:=value);
END_METHOD

METHOD set_Enable_user_scale : BOOL
VAR_INPUT
	value	: BOOL;
END_VAR
set_Enable_user_scale:=_p_Enable_user_scale.set_value(value:=value);
END_METHOD

METHOD set_Enable_vendor_calibration : BOOL
VAR_INPUT
	value	: BOOL;
END_VAR
set_Enable_vendor_calibration:=_p_Enable_vendor_calibration.set_value(value:=value);
END_METHOD

METHOD set_Gain : BOOL
VAR_INPUT
	value	: DINT;
END_VAR
set_Gain:=_p_Gain.set_value(value:=value);
END_METHOD

METHOD set_Offset : BOOL
VAR_INPUT
	value	: INT;
END_VAR
set_Offset:=_p_Offset.set_value(value:=value);
END_METHOD

METHOD set_Presentation : BOOL
VAR_INPUT
	value	: ENU_DT0801EN03;
END_VAR
set_Presentation:=_p_Presentation.set_value(value:=INT_TO_USINT(value));
END_METHOD

METHOD set_User_calibration_gain : BOOL
VAR_INPUT
	value	: UINT;
END_VAR
set_User_calibration_gain:=_p_User_calibration_gain.set_value(value:=value);
END_METHOD

METHOD set_User_calibration_offset : BOOL
VAR_INPUT
	value	: INT;
END_VAR
set_User_calibration_offset:=_p_User_calibration_offset.set_value(value:=value);
END_METHOD

METHOD set_Watchdog : BOOL
VAR_INPUT
	value	: ENU_DT0800EN02;
END_VAR
set_Watchdog:=_p_Watchdog.set_value(value:=int_TO_USINT(value));
END_METHOD

PROPERTY terminal_value : int
SET
linear_adc_to_phy(
	physical_min	:= _physical_min, 
	physical_max	:= _physical_max, 
	adc_min			:= _adc_min, 
	adc_max			:= _adc_max, 
	adc_value		:= terminal_value, 
	physical_value	=> _rValue, 
	errId			=> _errId
);

linear_adc_to_phy(
	physical_min	:= 0, 
	physical_max	:= 100, 
	adc_min			:= REAL_TO_DINT(_min_value), 
	adc_max			:= REAL_TO_DINT(_max_value), 
	adc_value		:= REAL_TO_DINT(_rValue), 
	physical_value	=> _value, 
	errId			=> _errId
);
END_SET
END_PROPERTY

PROPERTY value : REAL
GET
value := _value;
END_GET
END_PROPERTY

PROPERTY wcState : bool
GET
wcState:=_wcState;
END_GET
SET
_wcState:=wcState;
END_SET
END_PROPERTY

END_FUNCTION_BLOCK

// ---- analog_output/voltage/EL4102.TcPOU
(**
This function block abstracts the Beckhoff EtherCAT terminal EL4102 (0…10 V, 16 Bit)
*)
FUNCTION_BLOCK EL4102 implements I_terminal_execution
VAR_INPUT
END_VAR
VAR_OUTPUT
	AO_Voltage_channel_1 		: I_AO_Voltage :=_ar_channels[1];
	AO_Voltage_channel_2 		: I_AO_Voltage :=_ar_channels[1];
END_VAR
VAR
	WcState_WcState			AT%I*: BOOL;
	InfoData_State			AT%I*: UINT;
	InfoData_AdsAddr_netId  AT%I*: AMSNETID;
	InfoData_AdsAddr_port 	AT%I*: WORD;
	
	Channel_1_Output         AT%Q*: INT;
	Channel_2_Output         AT%Q*: INT;
	
	_ar_channels : ARRAY[1..NUMBER_OF_CHANNELS] OF AO_Voltage_Channel[
		(adc_min:=ADC_MIN, adc_max:=ADC_MAX, physical_min:=PHYSICAL_MIN, physical_max:=PHYSICAL_MAX, channel_number:=1),
		(adc_min:=ADC_MIN, adc_max:=ADC_MAX, physical_min:=PHYSICAL_MIN, physical_max:=PHYSICAL_MAX, channel_number:=2)
    ];

	// ===============================================================================
	// CoE handling  
	// ==============
    _I_CoE_com_handler      : I_CoE_communication_handler;
    _CoE_prop_handler       : CoE_property_handler;
    // ====  CoE properties  ===========
	_p_DeviceName 			: CoE_property_string(Index:=16#1008 , SubIndex:=0, writable:=FALSE, propertyType:=0, pollingInterval:=T#5S);
	_p_DeviceType 			: CoE_property_udint(Index:=16#1000 , SubIndex:=0, writable:=FALSE, propertyType:=0, pollingInterval:=T#5S);
	_p_ProductCode 			: CoE_property_udint(Index:=16#1018 , SubIndex:=2, writable:=FALSE, propertyType:=0, pollingInterval:=T#5S);
	_p_Revision 			: CoE_property_udint(Index:=16#1018 , SubIndex:=3, writable:=FALSE, propertyType:=0, pollingInterval:=T#5S);
	_p_SerialNumber 		: CoE_property_udint(Index:=16#1018 , SubIndex:=4, writable:=FALSE, propertyType:=0, pollingInterval:=T#5S);
	_p_SoftwareVersion		: CoE_property_string(Index:=16#100A , SubIndex:=0, writable:=FALSE, propertyType:=0, pollingInterval:=T#5S);
	_p_VendorId 			: CoE_property_udint(Index:=16#1018 , SubIndex:=1, writable:=FALSE, propertyType:=0, pollingInterval:=T#5S);
	_p_HardwareVersion		: CoE_property_string(Index:=16#1009 , SubIndex:=0, writable:=FALSE, propertyType:=0, pollingInterval:=T#5S);
	// ==============
	_properties  : ARRAY[1..8]OF I_CoE_property:=[
		_p_DeviceName, _p_DeviceType, _p_ProductCode, _p_Revision, _p_SerialNumber, 
		_p_SoftwareVersion, _p_VendorId, _p_HardwareVersion
	];
	// ===============================================================================
    
	_I_InterfaceManager : I_InterfaceManager;
    _terminal_name      : STRING;
    _terminal_id        : UINT;
    errId               : HAL_ErrorEnum;
	neg_wcState         : f_trig;
    _j                  : USINT;
END_VAR
VAR CONSTANT
	ADC_MIN        	: INT:=0;
	ADC_MAX        	: INT:=32767;
	PHYSICAL_MIN 	: INT:=0;
	PHYSICAL_MAX 	: INT:=10;
	
    HARDWARE_REVSION : UINT:=19;
    NUMBER_OF_CHANNELS : USINT:=2;
END_VAR

_ar_channels[1].wcState:= WcState_WcState;
_ar_channels[2].wcState:= WcState_WcState;

_ar_channels[1](terminal_address:=InfoData_AdsAddr_port, CoE_communication_handler:=_I_CoE_com_handler);
_ar_channels[2](terminal_address:=InfoData_AdsAddr_port, CoE_communication_handler:=_I_CoE_com_handler);

Channel_1_Output := _ar_channels[1].terminal_value;
Channel_2_Output := _ar_channels[2].terminal_value;

IF  _I_InterfaceManager <> 0 AND 
    _I_CoE_com_handler <> 0
THEN
    FOR _j:=1 TO NUMBER_OF_CHANNELS DO
        // should be possible to get rid of the address input 
        _ar_channels[_j](terminal_address:=InfoData_AdsAddr_port, CoE_communication_handler:=_I_CoE_com_handler);
    END_FOR
    
    _CoE_prop_handler(terminal_address:=InfoData_AdsAddr_port, CoE_communication_handler:=_I_CoE_com_handler, CoE_properties:=_properties);

    neg_wcState(CLK:=WcState_WcState);
    IF neg_wcState.Q THEN
        ;
    END_IF
END_IF

METHOD FB_init : BOOL
VAR_INPUT
	bInitRetains : BOOL; // if TRUE, the retain variables are initialized (warm start / cold start)
	bInCopyCode : BOOL;  // if TRUE, the instance afterwards gets moved into the copy code (online change)
	CoE_communication_handler : I_CoE_communication_handler;
    InterfaceManager            : I_InterfaceManager;
	name                        : STRING;
END_VAR

_I_CoE_com_handler := CoE_communication_handler;

FOR _j:=1 TO NUMBER_OF_CHANNELS DO
    _ar_channels[_j].CoE_communication_handler := CoE_communication_handler;
END_FOR

_terminal_name := name;
_I_InterfaceManager := InterfaceManager;

// register  terminal and all channel interfaces
IF InterfaceManager <> 0 THEN
    _I_InterfaceManager.register_terminal(terminal_name:=_terminal_name , errId=>errId , terminalId=>_terminal_id);
    
    FOR _j:=1 TO NUMBER_OF_CHANNELS DO
        _ar_channels[_j].register_channel(terminalId:=_terminal_id , I_interface_manager:=_I_InterfaceManager , errId=>errId );
        IF errId <> HAL_ErrorEnum.no_error THEN
            ;  // ToDo: add logging or Error handling 
        END_IF 
    END_FOR
END_IF
END_METHOD

METHOD run : BOOL
THIS^();
END_METHOD

END_FUNCTION_BLOCK

// ---- analog_output/voltage/EL4004.TcPOU
(**
This function block abstracts the Beckhoff EtherCAT terminal EL4004 (0…10 V, 12 Bit)
*)
FUNCTION_BLOCK EL4004 IMPLEMENTS I_terminal_execution
VAR_INPUT
END_VAR
VAR_OUTPUT
	AO_Voltage_channel_1 		: I_AO_Voltage :=_ar_channels[1];
	AO_Voltage_channel_2 		: I_AO_Voltage :=_ar_channels[2];
	AO_Voltage_channel_3 		: I_AO_Voltage :=_ar_channels[3];
	AO_Voltage_channel_4 		: I_AO_Voltage :=_ar_channels[4];
END_VAR
VAR
	WcState_WcState			AT%I*: BOOL;
	InfoData_State			AT%I*: UINT;
	InfoData_AdsAddr_netId  AT%I*: AMSNETID;
	InfoData_AdsAddr_port 	AT%I*: WORD;

	AO_Outputs_Channel_1_Analog_output         AT%Q*: INT;
	AO_Outputs_Channel_2_Analog_output         AT%Q*: INT;
	AO_Outputs_Channel_3_Analog_output         AT%Q*: INT;
	AO_Outputs_Channel_4_Analog_output         AT%Q*: INT;
	
	_ar_channels : ARRAY[1..NUMBER_OF_CHANNELS] OF AO_Voltage_Channel[
		(adc_min:=ADC_MIN, adc_max:=ADC_MAX, physical_min:=PHYSICAL_MIN, physical_max:=PHYSICAL_MAX, channel_number:=1),
		(adc_min:=ADC_MIN, adc_max:=ADC_MAX, physical_min:=PHYSICAL_MIN, physical_max:=PHYSICAL_MAX, channel_number:=2),
        (adc_min:=ADC_MIN, adc_max:=ADC_MAX, physical_min:=PHYSICAL_MIN, physical_max:=PHYSICAL_MAX, channel_number:=3),
        (adc_min:=ADC_MIN, adc_max:=ADC_MAX, physical_min:=PHYSICAL_MIN, physical_max:=PHYSICAL_MAX, channel_number:=4)
    ];
	// ===============================================================================
	// CoE handling  
	// ==============
    _I_CoE_com_handler      : I_CoE_communication_handler;
    _CoE_prop_handler       : CoE_property_handler;
    // ====  CoE properties  ===========
	_p_DeviceName 			: CoE_property_string(Index:=16#1008 , SubIndex:=0, writable:=FALSE, propertyType:=0, pollingInterval:=T#5S);
	_p_DeviceType 			: CoE_property_udint(Index:=16#1000 , SubIndex:=0, writable:=FALSE, propertyType:=0, pollingInterval:=T#5S);
	_p_ProductCode 			: CoE_property_udint(Index:=16#1018 , SubIndex:=2, writable:=FALSE, propertyType:=0, pollingInterval:=T#5S);
	_p_Revision 			: CoE_property_udint(Index:=16#1018 , SubIndex:=3, writable:=FALSE, propertyType:=0, pollingInterval:=T#5S);
	_p_SerialNumber 		: CoE_property_udint(Index:=16#1018 , SubIndex:=4, writable:=FALSE, propertyType:=0, pollingInterval:=T#5S);
	_p_SoftwareVersion		: CoE_property_string(Index:=16#100A , SubIndex:=0, writable:=FALSE, propertyType:=0, pollingInterval:=T#5S);
	_p_VendorId 			: CoE_property_udint(Index:=16#1018 , SubIndex:=1, writable:=FALSE, propertyType:=0, pollingInterval:=T#5S);
	_p_HardwareVersion		: CoE_property_string(Index:=16#1009 , SubIndex:=0, writable:=FALSE, propertyType:=0, pollingInterval:=T#5S);
	// ==============
	_properties  : ARRAY[1..8]OF I_CoE_property:=[
		_p_DeviceName, _p_DeviceType, _p_ProductCode, _p_Revision, _p_SerialNumber, 
		_p_SoftwareVersion, _p_VendorId, _p_HardwareVersion
	];
	// ===============================================================================
    
	_I_InterfaceManager : I_InterfaceManager;
    _terminal_name      : STRING;
    _terminal_id        : UINT;
    errId               : HAL_ErrorEnum;
	neg_wcState         : f_trig;
    _j                  : USINT;
END_VAR
VAR CONSTANT
	ADC_MIN        	: INT:=0;
	ADC_MAX        	: INT:=32767;
	PHYSICAL_MIN 	: INT:=0;
	PHYSICAL_MAX 	: INT:=10;
	
    HARDWARE_REVSION : UINT:=19;
    NUMBER_OF_CHANNELS : USINT:=4;
END_VAR


_ar_channels[1].wcState:= WcState_WcState;
_ar_channels[2].wcState:= WcState_WcState;
_ar_channels[3].wcState:= WcState_WcState;
_ar_channels[4].wcState:= WcState_WcState;

_ar_channels[1](terminal_address:=InfoData_AdsAddr_port, CoE_communication_handler:=_I_CoE_com_handler);
_ar_channels[2](terminal_address:=InfoData_AdsAddr_port, CoE_communication_handler:=_I_CoE_com_handler);
_ar_channels[3](terminal_address:=InfoData_AdsAddr_port, CoE_communication_handler:=_I_CoE_com_handler);
_ar_channels[4](terminal_address:=InfoData_AdsAddr_port, CoE_communication_handler:=_I_CoE_com_handler);

AO_Outputs_Channel_1_Analog_output := _ar_channels[1].terminal_value;
AO_Outputs_Channel_2_Analog_output := _ar_channels[2].terminal_value;
AO_Outputs_Channel_1_Analog_output := _ar_channels[3].terminal_value;
AO_Outputs_Channel_2_Analog_output := _ar_channels[4].terminal_value;

IF  _I_InterfaceManager <> 0 AND 
    _I_CoE_com_handler <> 0
THEN
    FOR _j:=1 TO NUMBER_OF_CHANNELS DO
        // should be possible to get rid of the address input 
        _ar_channels[_j](terminal_address:=InfoData_AdsAddr_port, CoE_communication_handler:=_I_CoE_com_handler);
    END_FOR
    
    _CoE_prop_handler(terminal_address:=InfoData_AdsAddr_port, CoE_communication_handler:=_I_CoE_com_handler, CoE_properties:=_properties);

    neg_wcState(CLK:=WcState_WcState);
    IF neg_wcState.Q THEN
        ;
    END_IF
END_IF

METHOD FB_init : BOOL
VAR_INPUT
	bInitRetains : BOOL; // if TRUE, the retain variables are initialized (warm start / cold start)
	bInCopyCode : BOOL;  // if TRUE, the instance afterwards gets moved into the copy code (online change)
	CoE_communication_handler: I_CoE_communication_handler;
    InterfaceManager            : I_InterfaceManager;
	name                        : STRING;
END_VAR

_I_CoE_com_handler := CoE_communication_handler;

FOR _j:=1 TO NUMBER_OF_CHANNELS DO
    _ar_channels[_j].CoE_communication_handler := CoE_communication_handler;
END_FOR

_terminal_name := name;
_I_InterfaceManager := InterfaceManager;

// register  terminal and all channel interfaces
IF InterfaceManager <> 0 THEN
    _I_InterfaceManager.register_terminal(terminal_name:=_terminal_name , errId=>errId , terminalId=>_terminal_id);
    
    FOR _j:=1 TO NUMBER_OF_CHANNELS DO
        _ar_channels[_j].register_channel(terminalId:=_terminal_id , I_interface_manager:=_I_InterfaceManager , errId=>errId );
        IF errId <> HAL_ErrorEnum.no_error THEN
            ;  // ToDo: add logging or Error handling 
        END_IF 
    END_FOR
END_IF
END_METHOD

METHOD run : BOOL
VAR_INPUT
END_VAR
THIS^();
END_METHOD

END_FUNCTION_BLOCK

// ---- analog_output/voltage/EL4134.TcPOU
(**
This function block abstracts the Beckhoff EtherCAT terminal EL4134 (-10…10 V, 16 Bit)
*)
FUNCTION_BLOCK EL4134 IMPLEMENTS I_terminal_execution
VAR_INPUT
END_VAR
VAR_OUTPUT
	AO_Voltage_channel_1 		: I_AO_Voltage :=_ar_channels[1];
	AO_Voltage_channel_2 		: I_AO_Voltage :=_ar_channels[2];
	AO_Voltage_channel_3 		: I_AO_Voltage :=_ar_channels[3];
	AO_Voltage_channel_4 		: I_AO_Voltage :=_ar_channels[4];
END_VAR
VAR
	WcState_WcState			AT%I*: BOOL;
	InfoData_State			AT%I*: UINT;
	InfoData_AdsAddr_netId  AT%I*: AMSNETID;
	InfoData_AdsAddr_port 	AT%I*: WORD;
	
	AO_Output_Channel_1_Analog_output         AT%Q*: INT;
	AO_Output_Channel_2_Analog_output         AT%Q*: INT;
	AO_Output_Channel_3_Analog_output         AT%Q*: INT;
	AO_Output_Channel_4_Analog_output         AT%Q*: INT;	

	_ar_channels : ARRAY[1..NUMBER_OF_CHANNELS] OF AO_Voltage_Channel[
		(adc_min:=ADC_MIN, adc_max:=ADC_MAX, physical_min:=PHYSICAL_MIN, physical_max:=PHYSICAL_MAX, channel_number:=1),
		(adc_min:=ADC_MIN, adc_max:=ADC_MAX, physical_min:=PHYSICAL_MIN, physical_max:=PHYSICAL_MAX, channel_number:=2),
        (adc_min:=ADC_MIN, adc_max:=ADC_MAX, physical_min:=PHYSICAL_MIN, physical_max:=PHYSICAL_MAX, channel_number:=3),
        (adc_min:=ADC_MIN, adc_max:=ADC_MAX, physical_min:=PHYSICAL_MIN, physical_max:=PHYSICAL_MAX, channel_number:=4)
    ];
    
	// ===============================================================================
	// CoE handling  
	// ==============
    _I_CoE_com_handler      : I_CoE_communication_handler;
    _CoE_prop_handler       : CoE_property_handler;
    // ====  CoE properties  ===========
	_p_DeviceName 			: CoE_property_string(Index:=16#1008 , SubIndex:=0, writable:=FALSE, propertyType:=0, pollingInterval:=T#5S);
	_p_DeviceType 			: CoE_property_udint(Index:=16#1000 , SubIndex:=0, writable:=FALSE, propertyType:=0, pollingInterval:=T#5S);
	_p_ProductCode 			: CoE_property_udint(Index:=16#1018 , SubIndex:=2, writable:=FALSE, propertyType:=0, pollingInterval:=T#5S);
	_p_Revision 			: CoE_property_udint(Index:=16#1018 , SubIndex:=3, writable:=FALSE, propertyType:=0, pollingInterval:=T#5S);
	_p_SerialNumber 		: CoE_property_udint(Index:=16#1018 , SubIndex:=4, writable:=FALSE, propertyType:=0, pollingInterval:=T#5S);
	_p_SoftwareVersion		: CoE_property_string(Index:=16#100A , SubIndex:=0, writable:=FALSE, propertyType:=0, pollingInterval:=T#5S);
	_p_VendorId 			: CoE_property_udint(Index:=16#1018 , SubIndex:=1, writable:=FALSE, propertyType:=0, pollingInterval:=T#5S);
	_p_HardwareVersion		: CoE_property_string(Index:=16#1009 , SubIndex:=0, writable:=FALSE, propertyType:=0, pollingInterval:=T#5S);
	// ==============
	_properties  : ARRAY[1..8]OF I_CoE_property:=[
		_p_DeviceName, _p_DeviceType, _p_ProductCode, _p_Revision, _p_SerialNumber, 
		_p_SoftwareVersion, _p_VendorId, _p_HardwareVersion
	];
	// ===============================================================================
    
	_I_InterfaceManager : I_InterfaceManager;
    _terminal_name      : STRING;
    _terminal_id        : UINT;
    errId               : HAL_ErrorEnum;
	neg_wcState         : f_trig;
    _j                  : USINT;
END_VAR
VAR CONSTANT
	ADC_MIN        	: INT:=-32767;
	ADC_MAX        	: INT:=32767;
	PHYSICAL_MIN 	: INT:=-10;
	PHYSICAL_MAX 	: INT:=10;
	
    HARDWARE_REVSION : UINT:=19;
    NUMBER_OF_CHANNELS : USINT:=4;
END_VAR


_ar_channels[1].wcState:= WcState_WcState;
_ar_channels[2].wcState:= WcState_WcState;
_ar_channels[3].wcState:= WcState_WcState;
_ar_channels[4].wcState:= WcState_WcState;

_ar_channels[1](terminal_address:=InfoData_AdsAddr_port, CoE_communication_handler:=_I_CoE_com_handler);
_ar_channels[2](terminal_address:=InfoData_AdsAddr_port, CoE_communication_handler:=_I_CoE_com_handler);
_ar_channels[3](terminal_address:=InfoData_AdsAddr_port, CoE_communication_handler:=_I_CoE_com_handler);
_ar_channels[4](terminal_address:=InfoData_AdsAddr_port, CoE_communication_handler:=_I_CoE_com_handler);

AO_Output_Channel_1_Analog_output := _ar_channels[1].terminal_value;
AO_Output_Channel_2_Analog_output := _ar_channels[2].terminal_value;
AO_Output_Channel_3_Analog_output := _ar_channels[3].terminal_value;
AO_Output_Channel_4_Analog_output := _ar_channels[4].terminal_value;

IF  _I_InterfaceManager <> 0 AND 
    _I_CoE_com_handler <> 0
THEN
    FOR _j:=1 TO NUMBER_OF_CHANNELS DO
        // should be possible to get rid of the address input 
        _ar_channels[_j](terminal_address:=InfoData_AdsAddr_port, CoE_communication_handler:=_I_CoE_com_handler);
    END_FOR
    
    _CoE_prop_handler(terminal_address:=InfoData_AdsAddr_port, CoE_communication_handler:=_I_CoE_com_handler, CoE_properties:=_properties);

    neg_wcState(CLK:=WcState_WcState);
    IF neg_wcState.Q THEN
        ;
    END_IF
END_IF

METHOD FB_init : BOOL
VAR_INPUT
	bInitRetains : BOOL; // if TRUE, the retain variables are initialized (warm start / cold start)
	bInCopyCode : BOOL;  // if TRUE, the instance afterwards gets moved into the copy code (online change)
	CoE_communication_handler : I_CoE_communication_handler;
    InterfaceManager            : I_InterfaceManager;
	name                        : STRING;
END_VAR

_I_CoE_com_handler := CoE_communication_handler;

FOR _j:=1 TO NUMBER_OF_CHANNELS DO
    _ar_channels[_j].CoE_communication_handler := CoE_communication_handler;
END_FOR

_terminal_name := name;
_I_InterfaceManager := InterfaceManager;

// register  terminal and all channel interfaces
IF InterfaceManager <> 0 THEN
    _I_InterfaceManager.register_terminal(terminal_name:=_terminal_name , errId=>errId , terminalId=>_terminal_id);
    
    FOR _j:=1 TO NUMBER_OF_CHANNELS DO
        _ar_channels[_j].register_channel(terminalId:=_terminal_id , I_interface_manager:=_I_InterfaceManager , errId=>errId );
        IF errId <> HAL_ErrorEnum.no_error THEN
            ;  // ToDo: add logging or Error handling 
        END_IF 
    END_FOR
END_IF
END_METHOD

METHOD run : BOOL
VAR_INPUT
END_VAR
THIS^();
END_METHOD

END_FUNCTION_BLOCK

// ---- coupler/EK1101.TcPOU
(**
	This function block abstracts the EtherCAT coupler EK1101.
	All inputs of this coupler should be linked to the function block.
	Terminals that are connected to the coupler should be abstracted with the according function blocks and
	passed into this function block to be executed, based on the state of the coupler and the sync_unit_ok, 
	which should be provided by the calling program.
*)
FUNCTION_BLOCK EK1101 IMPLEMENTS I_terminal_execution
VAR
	ID_ID					AT%I*: UINT;
	WcState_WcState			AT%I*: BOOL;
	WcState_InputToggle		AT%I*: BOOL;
	InfoData_State			AT%I*: UINT;
	
	_i				: DINT;
	_sync_unit_ok	: BOOL;
END_VAR
VAR_IN_OUT
	terminals: ARRAY[*] OF I_terminal_execution;
END_VAR


IF WcState_WcState  AND  _sync_unit_ok THEN
	FOR _i:=LOWER_BOUND(terminals, 1) TO UPPER_BOUND(terminals, 1) DO
		terminals[_i].run();
	END_FOR
ELSE
	// ToDo: put terminals in sync unit error state
	;
END_IF

METHOD FB_init : BOOL
VAR_INPUT
	bInitRetains : BOOL; // if TRUE, the retain variables are initialized (warm start / cold start)
	bInCopyCode : BOOL;  // if TRUE, the instance afterwards gets moved into the copy code (online change)
	CoE_communication_handler   : I_CoE_communication_handler;
	InterfaceManager            : I_InterfaceManager;
	name                        : STRING;
END_VAR
;
END_METHOD

METHOD run : BOOL
(*
VAR_INPUT
	sync_unit_ok	: BOOL;
END_VAR
*)
//THIS^._sync_unit_ok := sync_unit_ok;
THIS^();
END_METHOD

END_FUNCTION_BLOCK

// ---- digital_input/EL1008.TcPOU
(**
This function block abstracts the Beckhoff EtherCAT terminal EL1008
*)
FUNCTION_BLOCK EL1008 IMPLEMENTS I_terminal_execution
VAR_INPUT
END_VAR
VAR_OUTPUT
	DI_channel_1 		: I_HAL_DI :=_channel_1;
	DI_channel_2 		: I_HAL_DI :=_channel_2;
	DI_channel_3 		: I_HAL_DI :=_channel_3;
	DI_channel_4 		: I_HAL_DI :=_channel_4;
	DI_channel_5 		: I_HAL_DI :=_channel_5;
	DI_channel_6 		: I_HAL_DI :=_channel_6;
	DI_channel_7 		: I_HAL_DI :=_channel_7;
	DI_channel_8 		: I_HAL_DI :=_channel_8;
END_VAR
VAR
	WcState_WcState			AT%I*: BOOL;
	WcState_InputToggle		AT%I*: BOOL;
	InfoData_State			AT%I*: UINT;
	
	Channel_1_Input         AT%I*: BOOL;
	Channel_2_Input         AT%I*: BOOL;
	Channel_3_Input         AT%I*: BOOL;
	Channel_4_Input         AT%I*: BOOL;
	Channel_5_Input         AT%I*: BOOL;
	Channel_6_Input         AT%I*: BOOL;
	Channel_7_Input         AT%I*: BOOL;
	Channel_8_Input         AT%I*: BOOL;
	
	_channel_1 : HAL_DI_Channel(channel_number:=1);
	_channel_2 : HAL_DI_Channel(channel_number:=2);
	_channel_3 : HAL_DI_Channel(channel_number:=3);
	_channel_4 : HAL_DI_Channel(channel_number:=4);
	_channel_5 : HAL_DI_Channel(channel_number:=5);
	_channel_6 : HAL_DI_Channel(channel_number:=6);
	_channel_7 : HAL_DI_Channel(channel_number:=7);
	_channel_8 : HAL_DI_Channel(channel_number:=8);
END_VAR
VAR CONSTANT	
    HARDWARE_REVSION : UINT:=19;
END_VAR


_channel_1.wcState:= NOT  WcState_WcState;
_channel_2.wcState:= NOT  WcState_WcState;
_channel_3.wcState:= NOT  WcState_WcState;
_channel_4.wcState:= NOT  WcState_WcState;
_channel_5.wcState:= NOT  WcState_WcState;
_channel_6.wcState:= NOT  WcState_WcState;
_channel_7.wcState:= NOT  WcState_WcState;
_channel_8.wcState:= NOT  WcState_WcState;

_channel_1();
_channel_2();
_channel_3();
_channel_4();
_channel_5();
_channel_6();
_channel_7();
_channel_8();

_channel_1.terminal_value:=Channel_1_Input;
_channel_2.terminal_value:=Channel_2_Input;
_channel_3.terminal_value:=Channel_3_Input;
_channel_4.terminal_value:=Channel_4_Input;
_channel_5.terminal_value:=Channel_5_Input;
_channel_6.terminal_value:=Channel_6_Input;
_channel_7.terminal_value:=Channel_7_Input;
_channel_8.terminal_value:=Channel_8_Input;

METHOD FB_init : BOOL
VAR_INPUT
	bInitRetains : BOOL; // if TRUE, the retain variables are initialized (warm start / cold start)
	bInCopyCode : BOOL;  // if TRUE, the instance afterwards gets moved into the copy code (online change)
	CoE_communication_handler: I_CoE_communication_handler;
END_VAR
END_METHOD

METHOD run : BOOL
VAR_INPUT
END_VAR
THIS^();
END_METHOD

END_FUNCTION_BLOCK

// ---- digital_input/EL1104.TcPOU
(**
This function block abstracts the Beckhoff EtherCAT terminal EL1104
*)
FUNCTION_BLOCK EL1104 IMPLEMENTS I_terminal_execution
VAR_INPUT
END_VAR
VAR_OUTPUT
	DI_channel_1 		: I_HAL_DI :=_channel_1;
	DI_channel_2 		: I_HAL_DI :=_channel_2;
	DI_channel_3 		: I_HAL_DI :=_channel_3;
	DI_channel_4 		: I_HAL_DI :=_channel_4;
END_VAR
VAR
	WcState_WcState			AT%I*: BOOL;
	WcState_InputToggle		AT%I*: BOOL;
	InfoData_State			AT%I*: UINT;
	
	Channel_1_Input         AT%I*: BOOL;
	Channel_2_Input         AT%I*: BOOL;
	Channel_3_Input         AT%I*: BOOL;
	Channel_4_Input         AT%I*: BOOL;
	
	_channel_1 : HAL_DI_Channel(channel_number:=1);
	_channel_2 : HAL_DI_Channel(channel_number:=2);
	_channel_3 : HAL_DI_Channel(channel_number:=3);
	_channel_4 : HAL_DI_Channel(channel_number:=4);
END_VAR
VAR CONSTANT	
    HARDWARE_REVSION : UINT:=19;
END_VAR


_channel_1.wcState:= NOT  WcState_WcState;
_channel_2.wcState:= NOT  WcState_WcState;
_channel_3.wcState:= NOT  WcState_WcState;
_channel_4.wcState:= NOT  WcState_WcState;

_channel_1();
_channel_2();
_channel_3();
_channel_4();

_channel_1.terminal_value:=Channel_1_Input;
_channel_2.terminal_value:=Channel_2_Input;
_channel_3.terminal_value:=Channel_3_Input;
_channel_4.terminal_value:=Channel_4_Input;

METHOD FB_init : BOOL
VAR_INPUT
	bInitRetains : BOOL; // if TRUE, the retain variables are initialized (warm start / cold start)
	bInCopyCode : BOOL;  // if TRUE, the instance afterwards gets moved into the copy code (online change)
	CoE_communication_handler: I_CoE_communication_handler;
END_VAR
END_METHOD

METHOD run : BOOL
VAR_INPUT
END_VAR
THIS^();
END_METHOD

END_FUNCTION_BLOCK

// ---- digital_input/EL1144.TcPOU
(**
This function block abstracts the Beckhoff EtherCAT terminal EL1144
*)
FUNCTION_BLOCK EL1144 IMPLEMENTS I_terminal_execution
VAR_INPUT
END_VAR
VAR_OUTPUT
	DI_channel_1 		: I_HAL_DI :=_channel_1;
	DI_channel_2 		: I_HAL_DI :=_channel_2;
	DI_channel_3 		: I_HAL_DI :=_channel_3;
	DI_channel_4 		: I_HAL_DI :=_channel_4;
END_VAR
VAR
	WcState_WcState			AT%I*: BOOL;
	WcState_InputToggle		AT%I*: BOOL;
	InfoData_State			AT%I*: UINT;
	
	Channel_1_Input         AT%I*: BOOL;
	Channel_2_Input         AT%I*: BOOL;
	Channel_3_Input         AT%I*: BOOL;
	Channel_4_Input         AT%I*: BOOL;
	
	_channel_1 : HAL_DI_Channel(channel_number:=1);
	_channel_2 : HAL_DI_Channel(channel_number:=2);
	_channel_3 : HAL_DI_Channel(channel_number:=3);
	_channel_4 : HAL_DI_Channel(channel_number:=4);
END_VAR
VAR CONSTANT	
    HARDWARE_REVSION : UINT:=19;
END_VAR


_channel_1.wcState:= NOT  WcState_WcState;
_channel_2.wcState:= NOT  WcState_WcState;
_channel_3.wcState:= NOT  WcState_WcState;
_channel_4.wcState:= NOT  WcState_WcState;

_channel_1();
_channel_2();
_channel_3();
_channel_4();

_channel_1.terminal_value:=Channel_1_Input;
_channel_2.terminal_value:=Channel_2_Input;
_channel_3.terminal_value:=Channel_3_Input;
_channel_4.terminal_value:=Channel_4_Input;

METHOD FB_init : BOOL
VAR_INPUT
	bInitRetains : BOOL; // if TRUE, the retain variables are initialized (warm start / cold start)
	bInCopyCode : BOOL;  // if TRUE, the instance afterwards gets moved into the copy code (online change)
	CoE_communication_handler: I_CoE_communication_handler;
END_VAR
END_METHOD

METHOD run : BOOL
VAR_INPUT
END_VAR
THIS^();
END_METHOD

END_FUNCTION_BLOCK

// ---- digital_input/EL1124.TcPOU
(**
This function block abstracts the Beckhoff EtherCAT terminal EL1124
*)
FUNCTION_BLOCK EL1124 IMPLEMENTS I_terminal_execution
VAR_INPUT
END_VAR
VAR_OUTPUT
	DI_channel_1 		: I_HAL_DI :=_channel_1;
	DI_channel_2 		: I_HAL_DI :=_channel_2;
	DI_channel_3 		: I_HAL_DI :=_channel_3;
	DI_channel_4 		: I_HAL_DI :=_channel_4;
END_VAR
VAR
	WcState_WcState			AT%I*: BOOL;
	WcState_InputToggle		AT%I*: BOOL;
	InfoData_State			AT%I*: UINT;
	
	Channel_1_Input         AT%I*: BOOL;
	Channel_2_Input         AT%I*: BOOL;
	Channel_3_Input         AT%I*: BOOL;
	Channel_4_Input         AT%I*: BOOL;
	
	_channel_1 : HAL_DI_Channel(channel_number:=1);
	_channel_2 : HAL_DI_Channel(channel_number:=2);
	_channel_3 : HAL_DI_Channel(channel_number:=3);
	_channel_4 : HAL_DI_Channel(channel_number:=4);
END_VAR
VAR CONSTANT	
    HARDWARE_REVSION : UINT:=19;
END_VAR


_channel_1.wcState:= NOT  WcState_WcState;
_channel_2.wcState:= NOT  WcState_WcState;
_channel_3.wcState:= NOT  WcState_WcState;
_channel_4.wcState:= NOT  WcState_WcState;

_channel_1();
_channel_2();
_channel_3();
_channel_4();

_channel_1.terminal_value:=Channel_1_Input;
_channel_2.terminal_value:=Channel_2_Input;
_channel_3.terminal_value:=Channel_3_Input;
_channel_4.terminal_value:=Channel_4_Input;

METHOD FB_init : BOOL
VAR_INPUT
	bInitRetains : BOOL; // if TRUE, the retain variables are initialized (warm start / cold start)
	bInCopyCode : BOOL;  // if TRUE, the instance afterwards gets moved into the copy code (online change)
	CoE_communication_handler: I_CoE_communication_handler;
END_VAR
END_METHOD

METHOD run : BOOL
VAR_INPUT
END_VAR
THIS^();
END_METHOD

END_FUNCTION_BLOCK

// ---- digital_input/EL1809.TcPOU
(**
This function block abstracts the Beckhoff EtherCAT terminal EL1809
*)
FUNCTION_BLOCK EL1809 IMPLEMENTS I_terminal_execution
VAR_INPUT
END_VAR
VAR_OUTPUT
	DI_channel_1 		: I_HAL_DI :=_channel_1;
	DI_channel_2 		: I_HAL_DI :=_channel_2;
	DI_channel_3 		: I_HAL_DI :=_channel_3;
	DI_channel_4 		: I_HAL_DI :=_channel_4;
	DI_channel_5 		: I_HAL_DI :=_channel_5;
	DI_channel_6 		: I_HAL_DI :=_channel_6;
	DI_channel_7 		: I_HAL_DI :=_channel_7;
	DI_channel_8 		: I_HAL_DI :=_channel_8;
	DI_channel_9 		: I_HAL_DI :=_channel_9;
	DI_channel_10 		: I_HAL_DI :=_channel_10;
	DI_channel_11 		: I_HAL_DI :=_channel_11;
	DI_channel_12 		: I_HAL_DI :=_channel_12;
	DI_channel_13		: I_HAL_DI :=_channel_13;
	DI_channel_14		: I_HAL_DI :=_channel_14;
	DI_channel_15		: I_HAL_DI :=_channel_15;
	DI_channel_16		: I_HAL_DI :=_channel_16;
END_VAR
VAR
	WcState_WcState			AT%I*: BOOL;
	WcState_InputToggle		AT%I*: BOOL;
	InfoData_State			AT%I*: UINT;
	
	Channel_1_Input         AT%I*: BOOL;
	Channel_2_Input         AT%I*: BOOL;
	Channel_3_Input         AT%I*: BOOL;
	Channel_4_Input         AT%I*: BOOL;
	Channel_5_Input         AT%I*: BOOL;
	Channel_6_Input         AT%I*: BOOL;
	Channel_7_Input         AT%I*: BOOL;
	Channel_8_Input         AT%I*: BOOL;
	Channel_9_Input         AT%I*: BOOL;
	Channel_10_Input         AT%I*: BOOL;
	Channel_11_Input         AT%I*: BOOL;
	Channel_12_Input         AT%I*: BOOL;
	Channel_13_Input         AT%I*: BOOL;
	Channel_14_Input         AT%I*: BOOL;
	Channel_15_Input         AT%I*: BOOL;
	Channel_16_Input         AT%I*: BOOL;
	
	_channel_1 : HAL_DI_Channel(channel_number:=1);
	_channel_2 : HAL_DI_Channel(channel_number:=2);
	_channel_3 : HAL_DI_Channel(channel_number:=3);
	_channel_4 : HAL_DI_Channel(channel_number:=4);
	_channel_5 : HAL_DI_Channel(channel_number:=5);
	_channel_6 : HAL_DI_Channel(channel_number:=6);
	_channel_7 : HAL_DI_Channel(channel_number:=7);
	_channel_8 : HAL_DI_Channel(channel_number:=8);
	_channel_9 : HAL_DI_Channel(channel_number:=9);
	_channel_10 : HAL_DI_Channel(channel_number:=10);
	_channel_11 : HAL_DI_Channel(channel_number:=11);
	_channel_12 : HAL_DI_Channel(channel_number:=12);
	_channel_13 : HAL_DI_Channel(channel_number:=13);
	_channel_14 : HAL_DI_Channel(channel_number:=14);
	_channel_15 : HAL_DI_Channel(channel_number:=15);
	_channel_16 : HAL_DI_Channel(channel_number:=16);
END_VAR
VAR CONSTANT	
    HARDWARE_REVSION : UINT:=19;
END_VAR


_channel_1.wcState:= NOT  WcState_WcState;
_channel_2.wcState:= NOT  WcState_WcState;
_channel_3.wcState:= NOT  WcState_WcState;
_channel_4.wcState:= NOT  WcState_WcState;
_channel_5.wcState:= NOT  WcState_WcState;
_channel_6.wcState:= NOT  WcState_WcState;
_channel_7.wcState:= NOT  WcState_WcState;
_channel_8.wcState:= NOT  WcState_WcState;
_channel_9.wcState:= NOT  WcState_WcState;
_channel_10.wcState:= NOT  WcState_WcState;
_channel_11.wcState:= NOT  WcState_WcState;
_channel_12.wcState:= NOT  WcState_WcState;
_channel_13.wcState:= NOT  WcState_WcState;
_channel_14.wcState:= NOT  WcState_WcState;
_channel_15.wcState:= NOT  WcState_WcState;
_channel_16.wcState:= NOT  WcState_WcState;

_channel_1();
_channel_2();
_channel_3();
_channel_4();
_channel_5();
_channel_6();
_channel_7();
_channel_8();
_channel_9();
_channel_10();
_channel_11();
_channel_12();
_channel_13();
_channel_14();
_channel_15();
_channel_16();

_channel_1.terminal_value:=Channel_1_Input;
_channel_2.terminal_value:=Channel_2_Input;
_channel_3.terminal_value:=Channel_3_Input;
_channel_4.terminal_value:=Channel_4_Input;
_channel_5.terminal_value:=Channel_5_Input;
_channel_6.terminal_value:=Channel_6_Input;
_channel_7.terminal_value:=Channel_7_Input;
_channel_8.terminal_value:=Channel_8_Input;
_channel_9.terminal_value:=Channel_9_Input;
_channel_10.terminal_value:=Channel_10_Input;
_channel_11.terminal_value:=Channel_11_Input;
_channel_12.terminal_value:=Channel_12_Input;
_channel_13.terminal_value:=Channel_13_Input;
_channel_14.terminal_value:=Channel_14_Input;
_channel_15.terminal_value:=Channel_15_Input;
_channel_16.terminal_value:=Channel_16_Input;

METHOD FB_init : BOOL
VAR_INPUT
	bInitRetains : BOOL; // if TRUE, the retain variables are initialized (warm start / cold start)
	bInCopyCode : BOOL;  // if TRUE, the instance afterwards gets moved into the copy code (online change)
	CoE_communication_handler: I_CoE_communication_handler;
END_VAR
END_METHOD

METHOD run : BOOL
VAR_INPUT
END_VAR
THIS^();
END_METHOD

END_FUNCTION_BLOCK

// ---- digital_output/EL2008.TcPOU
(**
This function block abstracts the Beckhoff EtherCAT terminal EL2008
*)
FUNCTION_BLOCK EL2008 IMPLEMENTS I_terminal_execution
VAR_INPUT
END_VAR
VAR_OUTPUT
	DO_channel_1 		: I_HAL_DO :=_channel_1;
	DO_channel_2 		: I_HAL_DO :=_channel_2;
	DO_channel_3 		: I_HAL_DO :=_channel_3;
	DO_channel_4 		: I_HAL_DO :=_channel_4;
	DO_channel_5 		: I_HAL_DO :=_channel_5;
	DO_channel_6 		: I_HAL_DO :=_channel_6;
	DO_channel_7 		: I_HAL_DO :=_channel_7;
	DO_channel_8 		: I_HAL_DO :=_channel_8;
END_VAR
VAR
	WcState_WcState			AT%I*: BOOL;
	InfoData_State			AT%I*: UINT;
	
	Channel_1_Output         AT%Q*: BOOL;
	Channel_2_Output         AT%Q*: BOOL;
	Channel_3_Output         AT%Q*: BOOL;
	Channel_4_Output         AT%Q*: BOOL;
	Channel_5_Output         AT%Q*: BOOL;
	Channel_6_Output         AT%Q*: BOOL;
	Channel_7_Output         AT%Q*: BOOL;
	Channel_8_Output         AT%Q*: BOOL;
	
	_channel_1 : HAL_DO_Channel(channel_number:=1);
	_channel_2 : HAL_DO_Channel(channel_number:=2);
	_channel_3 : HAL_DO_Channel(channel_number:=3);
	_channel_4 : HAL_DO_Channel(channel_number:=4);
	_channel_5 : HAL_DO_Channel(channel_number:=5);
	_channel_6 : HAL_DO_Channel(channel_number:=6);
	_channel_7 : HAL_DO_Channel(channel_number:=7);
	_channel_8 : HAL_DO_Channel(channel_number:=8);
END_VAR
VAR CONSTANT	
    HARDWARE_REVSION : UINT:=19;
END_VAR


_channel_1.wcState:= NOT  WcState_WcState;
_channel_2.wcState:= NOT  WcState_WcState;
_channel_3.wcState:= NOT  WcState_WcState;
_channel_4.wcState:= NOT  WcState_WcState;
_channel_5.wcState:= NOT  WcState_WcState;
_channel_6.wcState:= NOT  WcState_WcState;
_channel_7.wcState:= NOT  WcState_WcState;
_channel_8.wcState:= NOT  WcState_WcState;

_channel_1();
_channel_2();
_channel_3();
_channel_4();
_channel_5();
_channel_6();
_channel_7();
_channel_8();

Channel_1_Output := _channel_1.terminal_value;
Channel_2_Output := _channel_2.terminal_value;
Channel_3_Output := _channel_3.terminal_value;
Channel_4_Output := _channel_4.terminal_value;
Channel_5_Output := _channel_5.terminal_value;
Channel_6_Output := _channel_6.terminal_value;
Channel_7_Output := _channel_7.terminal_value;
Channel_8_Output := _channel_8.terminal_value;

METHOD FB_init : BOOL
VAR_INPUT
	bInitRetains : BOOL; // if TRUE, the retain variables are initialized (warm start / cold start)
	bInCopyCode : BOOL;  // if TRUE, the instance afterwards gets moved into the copy code (online change)
	CoE_communication_handler: I_CoE_communication_handler;
END_VAR
END_METHOD

METHOD run : BOOL
VAR_INPUT
END_VAR
THIS^();
END_METHOD

END_FUNCTION_BLOCK

// ---- digital_output/EL2124.TcPOU
(**
This function block abstracts the Beckhoff EtherCAT terminal EL2124
*)
FUNCTION_BLOCK EL2124 IMPLEMENTS I_terminal_execution
VAR_INPUT
END_VAR
VAR_OUTPUT
	DO_channel_1 		: I_HAL_DO :=_channel_1;
	DO_channel_2 		: I_HAL_DO :=_channel_2;
	DO_channel_3 		: I_HAL_DO :=_channel_3;
	DO_channel_4 		: I_HAL_DO :=_channel_4;
END_VAR
VAR
	WcState_WcState			AT%I*: BOOL;
	InfoData_State			AT%I*: UINT;
	
	Channel_1_Output         AT%Q*: BOOL;
	Channel_2_Output         AT%Q*: BOOL;
	Channel_3_Output         AT%Q*: BOOL;
	Channel_4_Output         AT%Q*: BOOL;
	
	_channel_1 : HAL_DO_Channel(channel_number:=1);
	_channel_2 : HAL_DO_Channel(channel_number:=2);
	_channel_3 : HAL_DO_Channel(channel_number:=3);
	_channel_4 : HAL_DO_Channel(channel_number:=4);
END_VAR
VAR CONSTANT	
    HARDWARE_REVSION : UINT:=19;
END_VAR


_channel_1.wcState:= NOT  WcState_WcState;
_channel_2.wcState:= NOT  WcState_WcState;
_channel_3.wcState:= NOT  WcState_WcState;
_channel_4.wcState:= NOT  WcState_WcState;

_channel_1();
_channel_2();
_channel_3();
_channel_4();

Channel_1_Output := _channel_1.terminal_value;
Channel_2_Output := _channel_2.terminal_value;
Channel_3_Output := _channel_3.terminal_value;
Channel_4_Output := _channel_4.terminal_value;

METHOD FB_init : BOOL
VAR_INPUT
	bInitRetains : BOOL; // if TRUE, the retain variables are initialized (warm start / cold start)
	bInCopyCode : BOOL;  // if TRUE, the instance afterwards gets moved into the copy code (online change)
	CoE_communication_handler : I_CoE_communication_handler;
END_VAR
END_METHOD

METHOD run : BOOL
VAR_INPUT
END_VAR
THIS^();
END_METHOD

END_FUNCTION_BLOCK

// ---- digital_output/EL2024_0010.TcPOU
(**
This function block abstracts the Beckhoff EtherCAT terminal EL2024-0010
*)
FUNCTION_BLOCK EL2024_0010 IMPLEMENTS I_terminal_execution
VAR_INPUT
END_VAR
VAR_OUTPUT
	DO_channel_1 		: I_HAL_DO :=_channel_1;
	DO_channel_2 		: I_HAL_DO :=_channel_2;
	DO_channel_3 		: I_HAL_DO :=_channel_3;
	DO_channel_4 		: I_HAL_DO :=_channel_4;
END_VAR
VAR
	WcState_WcState			AT%I*: BOOL;
	InfoData_State			AT%I*: UINT;
	
	Channel_1_Output         AT%Q*: BOOL;
	Channel_2_Output         AT%Q*: BOOL;
	Channel_3_Output         AT%Q*: BOOL;
	Channel_4_Output         AT%Q*: BOOL;
	
	_channel_1 : HAL_DO_Channel(channel_number:=1);
	_channel_2 : HAL_DO_Channel(channel_number:=2);
	_channel_3 : HAL_DO_Channel(channel_number:=3);
	_channel_4 : HAL_DO_Channel(channel_number:=4);
END_VAR
VAR CONSTANT	
    HARDWARE_REVSION : UINT:=19;
END_VAR


_channel_1.wcState:= NOT  WcState_WcState;
_channel_2.wcState:= NOT  WcState_WcState;
_channel_3.wcState:= NOT  WcState_WcState;
_channel_4.wcState:= NOT  WcState_WcState;

_channel_1();
_channel_2();
_channel_3();
_channel_4();

Channel_1_Output := _channel_1.terminal_value;
Channel_2_Output := _channel_2.terminal_value;
Channel_3_Output := _channel_3.terminal_value;
Channel_4_Output := _channel_4.terminal_value;

METHOD FB_init : BOOL
VAR_INPUT
	bInitRetains : BOOL; // if TRUE, the retain variables are initialized (warm start / cold start)
	bInCopyCode : BOOL;  // if TRUE, the instance afterwards gets moved into the copy code (online change)
	CoE_communication_handler : I_CoE_communication_handler;
END_VAR
END_METHOD

METHOD run : BOOL
VAR_INPUT
END_VAR
THIS^();
END_METHOD

END_FUNCTION_BLOCK

// ---- digital_output/EL2502.TcPOU
(**
This function block abstracts the Beckhoff EtherCAT terminal EL2502
*)
FUNCTION_BLOCK EL2502 IMPLEMENTS I_terminal_execution
VAR_INPUT
END_VAR
VAR_OUTPUT
	DO_channel_1 		: I_HAL_DO :=_channel_1;
	DO_channel_2 		: I_HAL_DO :=_channel_2;
END_VAR
VAR
	WcState_WcState			AT%I*: BOOL;
	InfoData_State			AT%I*: UINT;
	InfoData_AdsAddr_netId  AT%I*: AMSNETID;
	InfoData_AdsAddr_port 	AT%I*: WORD;
	
	PWM_Outputs_Channel_1_PWM_output         AT%Q*: BOOL;
	PWM_Outputs_Channel_2_PWM_output         AT%Q*: BOOL;
	
	_channel_1 : HAL_DO_Channel(channel_number:=1);
	_channel_2 : HAL_DO_Channel(channel_number:=2);
END_VAR
VAR CONSTANT	
    HARDWARE_REVSION : UINT:=19;
END_VAR


_channel_1.wcState:= NOT  WcState_WcState;
_channel_2.wcState:= NOT  WcState_WcState;

_channel_1();
_channel_2();

Channel_1_Output := _channel_1.terminal_value;
Channel_2_Output := _channel_2.terminal_value;

METHOD FB_init : BOOL
VAR_INPUT
	bInitRetains : BOOL; // if TRUE, the retain variables are initialized (warm start / cold start)
	bInCopyCode : BOOL;  // if TRUE, the instance afterwards gets moved into the copy code (online change)
	CoE_communication_handler : I_CoE_property_handler;
END_VAR
END_METHOD

METHOD run : BOOL
VAR_INPUT
END_VAR
THIS^();
END_METHOD

END_FUNCTION_BLOCK

// ---- digital_output/EL2595.TcPOU
(**
This function block abstracts the Beckhoff EtherCAT terminal EL2595
*)
FUNCTION_BLOCK EL2595 IMPLEMENTS I_terminal_execution
VAR_INPUT
END_VAR
VAR_OUTPUT
	DO_channel_1 		: I_HAL_DO :=_channel_1;
END_VAR
VAR
	WcState_WcState			AT%I*: BOOL;
	WcState_InputToggle 	AT%I*: BOOL;
	InfoData_State			AT%I*: UINT;
	InfoData_AdsAddr_netId  AT%I*: AMSNETID;
	InfoData_AdsAddr_port 	AT%I*: WORD;
	
	DOX_Status_Status_Ready_to_activate      		AT%I*: BOOL;
	DOX_Status_Status_Output_active					AT%I*: BOOL;
	DOX_Status_Status_Switching_operation_counter   AT%I*: BOOL;
	DOX_Status_Status_Warning       				AT%I*: BOOL;
	DOX_Status_Status_Error       					AT%I*: BOOL;
	DOX_Status_Status_Digital_input       			AT%I*: BOOL;
	DOX_Status_Status_TxPDO_Toggle     				AT%I*: BOOL;
	DOX_Control_Control_Output     					AT%Q*: BOOL;
	DOX_Control_Control_Input_trigger_enable     	AT%Q*: BOOL;
	DOX_Control_Control_Reset     					AT%Q*: BOOL;
	
	_channel_1 : HAL_DO_Channel(channel_number:=1);
END_VAR
VAR CONSTANT	
    HARDWARE_REVSION : UINT:=19;
END_VAR


_channel_1.wcState:= NOT  WcState_WcState;

_channel_1();

DOX_Control_Control_Output := _channel_1.terminal_value;

METHOD FB_init : BOOL
VAR_INPUT
	bInitRetains : BOOL; // if TRUE, the retain variables are initialized (warm start / cold start)
	bInCopyCode : BOOL;  // if TRUE, the instance afterwards gets moved into the copy code (online change)
	CoE_communication_handler : I_CoE_communication_handler;
END_VAR
END_METHOD

METHOD run : BOOL
VAR_INPUT
END_VAR
THIS^();
END_METHOD

END_FUNCTION_BLOCK

// ---- digital_output/EL2612.TcPOU
(**
This function block abstracts the Beckhoff EtherCAT terminal EL2612
*)
FUNCTION_BLOCK EL2612 IMPLEMENTS I_terminal_execution
VAR_INPUT
END_VAR
VAR_OUTPUT
	DO_channel_1 		: I_HAL_DO :=_channel_1;
	DO_channel_2 		: I_HAL_DO :=_channel_2;
END_VAR
VAR
	WcState_WcState			AT%I*: BOOL;
	InfoData_State			AT%I*: UINT;
	
	Channel_1_Output         AT%Q*: BOOL;
	Channel_2_Output         AT%Q*: BOOL;
	
	_channel_1 : HAL_DO_Channel(channel_number:=1);
	_channel_2 : HAL_DO_Channel(channel_number:=2);
END_VAR
VAR CONSTANT	
    HARDWARE_REVSION : UINT:=19;
END_VAR


_channel_1.wcState:= NOT  WcState_WcState;
_channel_2.wcState:= NOT  WcState_WcState;

_channel_1();
_channel_2();

Channel_1_Output := _channel_1.terminal_value;
Channel_2_Output := _channel_2.terminal_value;

METHOD FB_init : BOOL
VAR_INPUT
	bInitRetains : BOOL; // if TRUE, the retain variables are initialized (warm start / cold start)
	bInCopyCode : BOOL;  // if TRUE, the instance afterwards gets moved into the copy code (online change)
	CoE_communication_handler : I_CoE_communication_handler;
END_VAR
END_METHOD

METHOD run : BOOL
VAR_INPUT
END_VAR
THIS^();
END_METHOD

END_FUNCTION_BLOCK

// ---- digital_output/EL2521.TcPOU
(**
This function block abstracts the Beckhoff EtherCAT terminal EL2521
*)
FUNCTION_BLOCK EL2521 IMPLEMENTS I_terminal_execution
VAR_INPUT
END_VAR
VAR_OUTPUT
//	DO_channel_1 		: I_HAL_DO :=_channel_1;
END_VAR
VAR
	WcState_WcState			AT%I*: BOOL;
	InfoData_State			AT%I*: UINT;
	InfoData_AdsAddr_netId  AT%I*: AMSNETID;
	InfoData_AdsAddr_port 	AT%I*: WORD;
	
//	Channel_1_Output         AT%Q*: BOOL;
	
	_channel_1 : HAL_DO_Channel(channel_number:=1);
END_VAR
VAR CONSTANT	
    HARDWARE_REVSION : UINT:=19;
END_VAR


_channel_1.wcState:= NOT  WcState_WcState;

_channel_1();

Channel_1_Output := _channel_1.terminal_value;

METHOD FB_init : BOOL
VAR_INPUT
	bInitRetains : BOOL; // if TRUE, the retain variables are initialized (warm start / cold start)
	bInCopyCode : BOOL;  // if TRUE, the instance afterwards gets moved into the copy code (online change)
	CoE_communication_handler : I_CoE_property_handler;
END_VAR
END_METHOD

METHOD run : BOOL
VAR_INPUT
END_VAR
THIS^();
END_METHOD

END_FUNCTION_BLOCK

// ---- digital_output/EL2004.TcPOU
(**
This function block abstracts the Beckhoff EtherCAT terminal EL2004
*)
FUNCTION_BLOCK EL2004 IMPLEMENTS I_terminal_execution
VAR_INPUT
END_VAR
VAR_OUTPUT
	DO_channel_1 		: I_HAL_DO :=_channel_1;
	DO_channel_2 		: I_HAL_DO :=_channel_2;
	DO_channel_3 		: I_HAL_DO :=_channel_3;
	DO_channel_4 		: I_HAL_DO :=_channel_4;
END_VAR
VAR
	WcState_WcState			AT%I*: BOOL;
	InfoData_State			AT%I*: UINT;
	
	Channel_1_Output         AT%Q*: BOOL;
	Channel_2_Output         AT%Q*: BOOL;
	Channel_3_Output         AT%Q*: BOOL;
	Channel_4_Output         AT%Q*: BOOL;
	
	_channel_1 : HAL_DO_Channel(channel_number:=1);
	_channel_2 : HAL_DO_Channel(channel_number:=2);
	_channel_3 : HAL_DO_Channel(channel_number:=3);
	_channel_4 : HAL_DO_Channel(channel_number:=4);
END_VAR
VAR CONSTANT	
    HARDWARE_REVSION : UINT:=19;
END_VAR


_channel_1.wcState:= NOT  WcState_WcState;
_channel_2.wcState:= NOT  WcState_WcState;
_channel_3.wcState:= NOT  WcState_WcState;
_channel_4.wcState:= NOT  WcState_WcState;

_channel_1();
_channel_2();
_channel_3();
_channel_4();

Channel_1_Output := _channel_1.terminal_value;
Channel_2_Output := _channel_2.terminal_value;
Channel_3_Output := _channel_3.terminal_value;
Channel_4_Output := _channel_4.terminal_value;

METHOD FB_init : BOOL
VAR_INPUT
	bInitRetains : BOOL; // if TRUE, the retain variables are initialized (warm start / cold start)
	bInCopyCode : BOOL;  // if TRUE, the instance afterwards gets moved into the copy code (online change)
	CoE_communication_handler: I_CoE_communication_handler;
END_VAR
END_METHOD

METHOD run : BOOL
VAR_INPUT
END_VAR
THIS^();
END_METHOD

END_FUNCTION_BLOCK

// ---- digital_output/EL2634.TcPOU
(**
This function block abstracts the Beckhoff EtherCAT terminal EL2634
*)
FUNCTION_BLOCK EL2634 IMPLEMENTS I_terminal_execution
VAR_INPUT
END_VAR
VAR_OUTPUT
	DO_channel_1 		: I_HAL_DO :=_channel_1;
	DO_channel_2 		: I_HAL_DO :=_channel_2;
	DO_channel_3 		: I_HAL_DO :=_channel_3;
	DO_channel_4 		: I_HAL_DO :=_channel_4;
END_VAR
VAR
	WcState_WcState			AT%I*: BOOL;
	InfoData_State			AT%I*: UINT;
	
	Channel_1_Output         AT%Q*: BOOL;
	Channel_2_Output         AT%Q*: BOOL;
	Channel_3_Output         AT%Q*: BOOL;
	Channel_4_Output         AT%Q*: BOOL;
	
	_channel_1 : HAL_DO_Channel(channel_number:=1);
	_channel_2 : HAL_DO_Channel(channel_number:=2);
	_channel_3 : HAL_DO_Channel(channel_number:=3);
	_channel_4 : HAL_DO_Channel(channel_number:=4);
END_VAR
VAR CONSTANT	
    HARDWARE_REVSION : UINT:=19;
END_VAR


_channel_1.wcState:= NOT  WcState_WcState;
_channel_2.wcState:= NOT  WcState_WcState;
_channel_3.wcState:= NOT  WcState_WcState;
_channel_4.wcState:= NOT  WcState_WcState;

_channel_1();
_channel_2();
_channel_3();
_channel_4();

Channel_1_Output := _channel_1.terminal_value;
Channel_2_Output := _channel_2.terminal_value;
Channel_3_Output := _channel_3.terminal_value;
Channel_4_Output := _channel_4.terminal_value;

METHOD FB_init : BOOL
VAR_INPUT
	bInitRetains : BOOL; // if TRUE, the retain variables are initialized (warm start / cold start)
	bInCopyCode : BOOL;  // if TRUE, the instance afterwards gets moved into the copy code (online change)
	CoE_communication_handler : I_CoE_communication_handler;
END_VAR
END_METHOD

METHOD run : BOOL
VAR_INPUT
END_VAR
THIS^();
END_METHOD

END_FUNCTION_BLOCK

// ---- digital_output/EL2624.TcPOU
(**
This function block abstracts the Beckhoff EtherCAT terminal EL2624
*)
FUNCTION_BLOCK EL2624 IMPLEMENTS I_terminal_execution
VAR_INPUT
END_VAR
VAR_OUTPUT
	DO_channel_1 		: I_HAL_DO :=_channel_1;
	DO_channel_2 		: I_HAL_DO :=_channel_2;
	DO_channel_3 		: I_HAL_DO :=_channel_3;
	DO_channel_4 		: I_HAL_DO :=_channel_4;
END_VAR
VAR
	WcState_WcState			AT%I*: BOOL;
	InfoData_State			AT%I*: UINT;
	
	Channel_1_Output         AT%Q*: BOOL;
	Channel_2_Output         AT%Q*: BOOL;
	Channel_3_Output         AT%Q*: BOOL;
	Channel_4_Output         AT%Q*: BOOL;
	
	_channel_1 : HAL_DO_Channel(channel_number:=1);
	_channel_2 : HAL_DO_Channel(channel_number:=2);
	_channel_3 : HAL_DO_Channel(channel_number:=3);
	_channel_4 : HAL_DO_Channel(channel_number:=4);
END_VAR
VAR CONSTANT	
    HARDWARE_REVSION : UINT:=19;
END_VAR


_channel_1.wcState:= NOT  WcState_WcState;
_channel_2.wcState:= NOT  WcState_WcState;
_channel_3.wcState:= NOT  WcState_WcState;
_channel_4.wcState:= NOT  WcState_WcState;

_channel_1();
_channel_2();
_channel_3();
_channel_4();

Channel_1_Output := _channel_1.terminal_value;
Channel_2_Output := _channel_2.terminal_value;
Channel_3_Output := _channel_3.terminal_value;
Channel_4_Output := _channel_4.terminal_value;

METHOD FB_init : BOOL
VAR_INPUT
	bInitRetains : BOOL; // if TRUE, the retain variables are initialized (warm start / cold start)
	bInCopyCode : BOOL;  // if TRUE, the instance afterwards gets moved into the copy code (online change)
	CoE_communication_handler : I_CoE_communication_handler;
END_VAR
END_METHOD

METHOD run : BOOL
VAR_INPUT
END_VAR
THIS^();
END_METHOD

END_FUNCTION_BLOCK

// ---- digital_output/EL2794.TcPOU
(**
This function block abstracts the Beckhoff EtherCAT terminal EL2794
*)
FUNCTION_BLOCK EL2794 IMPLEMENTS I_terminal_execution
VAR_INPUT
END_VAR
VAR_OUTPUT
	DO_channel_1 		: I_HAL_DO :=_channel_1;
	DO_channel_2 		: I_HAL_DO :=_channel_2;
	DO_channel_3 		: I_HAL_DO :=_channel_3;
	DO_channel_4 		: I_HAL_DO :=_channel_4;
END_VAR
VAR
	WcState_WcState			AT%I*: BOOL;
	InfoData_State			AT%I*: UINT;
	
	Channel_1_Output         AT%Q*: BOOL;
	Channel_2_Output         AT%Q*: BOOL;
	Channel_3_Output         AT%Q*: BOOL;
	Channel_4_Output         AT%Q*: BOOL;
	
	_channel_1 : HAL_DO_Channel(channel_number:=1);
	_channel_2 : HAL_DO_Channel(channel_number:=2);
	_channel_3 : HAL_DO_Channel(channel_number:=3);
	_channel_4 : HAL_DO_Channel(channel_number:=4);
END_VAR
VAR CONSTANT	
    HARDWARE_REVSION : UINT:=19;
END_VAR


_channel_1.wcState:= NOT  WcState_WcState;
_channel_2.wcState:= NOT  WcState_WcState;
_channel_3.wcState:= NOT  WcState_WcState;
_channel_4.wcState:= NOT  WcState_WcState;

_channel_1();
_channel_2();
_channel_3();
_channel_4();

Channel_1_Output := _channel_1.terminal_value;
Channel_2_Output := _channel_2.terminal_value;
Channel_3_Output := _channel_3.terminal_value;
Channel_4_Output := _channel_4.terminal_value;

METHOD FB_init : BOOL
VAR_INPUT
	bInitRetains : BOOL; // if TRUE, the retain variables are initialized (warm start / cold start)
	bInCopyCode : BOOL;  // if TRUE, the instance afterwards gets moved into the copy code (online change)
	CoE_communication_handler : I_CoE_communication_handler;
END_VAR
END_METHOD

METHOD run : BOOL
VAR_INPUT
END_VAR
THIS^();
END_METHOD

END_FUNCTION_BLOCK

// ---- Project Information/F_GetCompany.TcPOU
// This function has been automatically generated from the project information.
{attribute 'signature_flag' := '1073741824'}
{attribute 'TcGenerated'}
{attribute 'no-analysis'}
FUNCTION F_GetCompany : WSTRING
VAR_INPUT
	
END_VAR

F_GetCompany := "none";

END_FUNCTION

// ---- Project Information/F_GetVersion.TcPOU
// This function has been automatically generated from the project information.
{attribute 'signature_flag' := '1073741824'}
{attribute 'TcGenerated'}
{attribute 'no-analysis'}
FUNCTION F_GetVersion : ST_LibVersion
VAR_INPUT
	
END_VAR

F_GetVersion.iMajor := 0;
F_GetVersion.iMinor := 1;
F_GetVersion.iBuild := 4;
F_GetVersion.iRevision := 0;

END_FUNCTION
